(* PLC project primary, CODESYS STW CODESYS V3.5 SP11 - ESX-3CS, author Isoloader *)
(* stored: creationDateTime 2026-05-19T11:23:56.1136893, version 0.101, modificationDateTime 2026-05-14T13:26:08.1458645, organization Isoloader *)

(* {attribute 'strict'} *)
{attribute 'qualified_only'}
TYPE t_bms_fault_id : (cBMSFaultCellOverVoltageAlarmWarning := 1, cBMSFaultCellOverVoltageAlarmCritical := 2, cBMSFaultCellOverVoltageAlarmSevere := 3, cBMSFaultCellUnderVoltageAlarmWarning := 4, cBMSFaultCellUnderVoltageAlarmCritical := 5, cBMSFaultCellUnderVoltageAlarmSevere := 6, cBMSFaultCellOverDischargeAlarm := 7, cBMSFaultSystemOverVoltageAlarmWarning := 8, cBMSFaultSystemOverVoltageAlarmCritical := 9, cBMSFaultSystemOvervoltageAlarmSevere := 10, cBMSFaultSystemUnderVoltageAlarmWarning := 11, cBMSFaultSystemUnderVoltageAlarmCritical := 12, cBMSFaultSystemUnderVoltageAlarmSevere := 13, cBMSFaultCellHighTemperatureAlarmWarning := 14, cBMSFaultCellHighTemperatureAlarmCritical := 15, cBMSFaultCellHighTemperatureAlarmSevere := 16, cBMSFaultCellLowTemperatureAlarm := 17, cBMSFaultTemperatureDifferenceisTooLargeAlarmWarning := 18, cBMSFaultTemperatureDifferenceisTooLargeAlarmCritical := 19, cBMSFaultTemperatureDifferenceisTooLargeAlarmSevere := 20, cBMSFaultFireAlarm := 21, cBMSFaultPulseDischargeOverCurrentAlarmWarning := 22, cBMSFaultPulseDischargeOverCurrentAlarmCritical := 23, cBMSFaultPulseDischargeOverCurrentAlarmSevere := 24, cBMSFaultPulseRechargeOverCurrentAlarmWarning := 25, cBMSFaultPulseRechargeOverCurrentAlarmCritical := 26, cBMSFaultPulseRechargeOverCurrentAlarmSevere := 27, cBMSFaultCurrentSensorFaultAlarm := 28, cBMSFaultBMSLowVoltagePowerSupplyisAbnormalAlarm := 29, cBMSFaultSOCDifferenceisTooLargeAlarm := 30, cBMSFaultSOCJumpFaultAlarm := 31, cBMSFaultLowSOCAlarmWarning := 32, cBMSFaultLowSOCAlarmCritical := 33, cBMSFaultLowSOCAlarmSevere := 34, cBMSFaultThermalManagementSystemFaultAlarm := 35, cBMSFaultPackSelfProtectionAlarm := 37, cBMSFaultMainCircuitPrechargePrecheckFaultAlarm := 38, cBMSFaultLowInsulationInDrivingAlarmWarning := 40, cBMSFaultLowInsulationInDrivingAlarmCritical := 41, cBMSFaultLowInsulationInDrivingAlarmSevere := 42, cBMSFaultLowInsulationInChargingAlarm := 43, cBMSFaultACANCommunicationFaultAlarm := 44, cBMSFaultBMSInternalCommunicationFaultAlarm := 45, cBMSFaultBranchDisconnectedFaultAlarm := 47, cBMSFaultHVILFaultAlarm := 48, cBMSFaultMainPositiveRelayCannotbeClosedAlarm := 51, cBMSFaultMainPositiveRelayWeldedAlarm := 52, cBMSFaultMainNegativeRelayCannotbeClosedAlarm := 53, cBMSFaultMainNegativeRelayWeldedAlarm := 54, cBMSFaultChargeableEnergyStorageSystemMismatchAlarm := 72, cBMSFaultDischargingCurrentIsTooLargeInChargingAlarm := 73, cBMSFaultChargingCurrentIsTooLargeAlarm := 74, cBMSFaultFireAlarmDetectorFault := 79, cBMSFaultCellPoorConsistencyAlarm := 100, cBMSFaultSOCAlarmTooHigh := 101, cBMSFaultContinuousDischargeOvercurrentAlarmWarning := 105, cBMSFaultContinuousDischargeOvercurrentAlarmCritical := 106, cBMSFaultContinuousDischargeOvercurrentAlarmSevere := 107);
END_TYPE

(* values of t_motor_emcy_id: cEMCY_PEV_NOT_OK: change from 65499, duplicate error; cEMCY_SP_MISMATCH_XX: cEMCY_SP_MISMATCH_PUMP := 65521,//change from 65521, duplicate; cEMCY_THROTTLE_PROG: cEMCY_OPEN_COIL_EV := 65522, //duplicate id *)

(* {attribute 'strict'} *)
{attribute 'qualified_only'}
TYPE t_motor_emcy_id : (cEMCY_none := 0, cEMCY_MC_EB_COIL_SHORT := 8784, cEMCY_STBY_HIGH := 8977, cEMCY_PUMP_ZERO_EVER := 8978, cEMCY_WRONG_SET_BAT := 12544, cEMCY_WRONG_KEY_VOLT := 12545, cEMCY_VMN_HIGH := 12560, cEMCY_INIT_VMN_HIGH := 12561, cEMCY_VMN_LOW := 12576, cEMCY_INIT_VMN_LOW := 12577, cEMCY_CAPACITOR_CHARGE := 12592, cEMCY_DRIVER_SHORTED := 12817, cEMCY_CONTACTOR_DRIVER := 12833, cEMCY_EB_DRIVSHRT := 12834, cEMCY_POS_EB_SHORTED := 12835, cEMCY_EB_DRIVOPEN := 12836, cEMCY_SMARTDRIVER_KO := 13058, cEMCY_EEPROM_KO := 13840, cEMCY_THERMIC_SENS_KO := 16913, cEMCY_SENS_MOT_TEMP_KO := 17169, cEMCY_AUX_BATT_SHORT := 20481, cEMCY_EVP_COIL_OPEN := 20482, cEMCY_EVP_DRIV_SHORT := 20483, cEMCY_EVP_COIL_SHORT := 20484, cEMCY_EVP2_COIL_OPEN := 20722, cEMCY_EVP2_DRIV_SHORT := 20723, cEMCY_EVP2_COIL_SHORT := 20724, cEMCY_VKEY_OFF_SHORTED := 20737, cEMCY_LOGIC_FAILURE_1 := 20756, cEMCY_CONTACTOR_OPEN := 21569, cEMCY_CONTACTOR_CLOSED := 21570, cEMCY_WATCHDOG := 24592, cEMCY_CURRENT_GAIN := 25346, cEMCY_NO_CAN_MSG := 33072, cEMCY_NO_CAN_WR_MSGXX := 33073, cEMCY_LOGIC_FAILURE_3 := 65297, cEMCY_LOGIC_FAILURE_2 := 65298, cEMCY_PUMP_VMN_LOW := 65308, cEMCY_PUMP_VMN_HIGH := 65309, cEMCY_BATTERY_LOW := 65346, cEMCY_VACC_NOT_OK := 65358, cEMCY_INCORRECT_START := 65359, cEMCY_FORW_BACK := 65360, cEMCY_WRONG_FBSENSSET := 65361, cEMCY_PEDAL_WIRE_KO := 65366, cEMCY_BACK_EMF_HIGH := 65418, cEMCY_THERMPUSENSKO := 65419, cEMCY_1175_NOT_ACTIVE := 65420, cEMCY_STO_SS1_ACTIVEXX := 65421, cEMCY_STO_SS1_ALARM_XX := 65422, cEMCY_SAFETY_INIT_XX := 65423, cEMCY_SAFETY_WARN_XX := 65424, cEMCY_SAFETY_SW_XX := 65425, cEMCY_SAFETY_DIAG_XX := 65426, cEMCY_BMS_FAULT := 65427, cEMCY_BMS_NOT_READY := 65428, cEMCY_WRONG_PERFORM := 65429, cEMCY_NO_CAN_MSG_DISP := 65430, cEMCY_POT_MISMATCH := 65431, cEMCY_SENSOR_SUPPLY_XX := 65432, cEMCY_OFFSET_SPDSENS := 65433, cEMCY_AGV := 65434, cEMCY_REMA_T_ALARM := 65436, cEMCY_FAULT_DRVPOWER := 65437, cEMCY_NOT_RDY_DRVPOW := 65438, cEMCY_HVIL_FAIL := 65439, cEMCY_SENS_BAT_TEMP_KO := 65440, cEMCY_RPM_HIGH := 65441, cEMCY_POSEBSHORT_PIN := 65442, cEMCY_ED_SLIP_MISMATCH := 65443, cEMCY_POSEBSHORT_GND := 65444, cEMCY_SHORT_CIRCUIT_KO := 65445, cEMCY_SHORT_CIRCUIT := 65446, cEMCY_IMS_ERROR := 65447, cEMCY_SPEED_FBERR_XX := 65448, cEMCY_EMERGENCY := 65449, cEMCY_SPEED_OVERHEAD := 65455, cEMCY_COIL_SHOR_EB := 65457, cEMCY_MOTOR_TEMP_STOP := 65458, cEMCY_STEER_SENSOR_KO := 65459, cEMCY_OVERLOAD := 65460, cEMCY_EVP2_DRIVER_OPEN := 65464, cEMCY_TILLER_ERROR := 65465, cEMCY_LIFT_LOWER := 65467, cEMCY_PUMP_VACC_NOT_OK := 65468, cEMCY_PUMP_INC_START := 65469, cEMCY_PUMP_VMN_NOT_OK := 65470, cEMCY_PUMP_I_NO_ZERO := 65471, cEMCY_PUMP_VACC_RANGE := 65472, cEMCY_MOTPHASE_SH := 65476, cEMCY_WRONG_SLAVE_VER := 65477, cEMCY_MS_PAR_CHK_MISM := 65478, cEMCY_PARAM_TRANSFER := 65479, cEMCY_VDC_OFF_SHORTED := 65480, cEMCY_CURRENT_PROFILE := 65481, cEMCY_VDC_LINK_OVERV := 65482, cEMCY_HW_FAULT_MC := 65483, cEMCY_BRAKE_RUN_OUT := 65484, cEMCY_EPS_RELAY_OPEN := 65485, cEMCY_WRONG_RAM_MEM := 65490, cEMCY_STALL_ROTOR := 65491, cEMCY_POWER_MISMATCH := 65492, cEMCY_WSET_TG_EB_XX := 65492, cEMCY_INPUT_MISMATCH := 65493, cEMCY_POSITIVE_LC_OPEN := 65493, cEMCY_EB_COIL_OPEN := 65496, cEMCY_PEB_PEVP_NOT_OK := 65499, cEMCY_PEV_NOT_OK := 65500, cEMCY_HANDBRAKE := 65501, cEMCY_SEAT_MISMATCH := 65502, cEMCY_VACC_OUT_RANGE := 65506, cEMCY_HW_FAULT := 65507, cEMCY_OUT_MISMATCH_XX := 65507, cEMCY_HW_FAULT_EB := 65509, cEMCY_LC_COIL_OPEN := 65510, cEMCY_CONT_DRV_EV := 65512, cEMCY_POWERMOS_SHORTED := 65513, cEMCY_CTRAP_THRESHOLD := 65515, cEMCY_HW_FAULT_EV := 65518, cEMCY_CONTROLLER_MISM := 65519, cEMCY_OUT_MISMATCH_PU := 65520, cEMCY_COIL_SHOR_EVAUX := 65521, cEMCY_SP_MISMATCH_XX := 65522, cEMCY_THROTTLE_PROG := 65523, cEMCY_IQ_MISMATCHED := 65525, cEMCY_EVP_DRIVER_OPEN := 65528, cEMCY_DRV_SHOR_EV := 65529, cEMCY_ANALOG_INPUT := 65530, cEMCY_FIELD_ORIENT_KO := 65533);
END_TYPE

TYPE t_radio_emcy_id : (cEMCY_none := 0, cEMCY_CAN_OVERRUN := 33040, cEMCY_CAN_IN_ERROR_PASSIVE_MODE := 33056, cEMCY_LIFE_GUARD_ERROR_OR_HEARTBEAT_ERROR := 33072, cEMCY_RECOVERED_FROM_BUS_OFF := 33088, cEMCY_TRANSMIT_COB_ID_COLLISION := 33104, cEMCY_PDO_NOT_PROCESSED_DUE_TO_LENGTH_ERROR := 33296, cEMCY_PDO_LENGTH_EXCEEDED := 33312, cEMCY_GENERIC_ERROR := 4096, cEMCY_CURRENT := 8192, cEMCY_CURRENT_DEVICE_INPUT_SIDE := 8448, cEMCY_CURRENT_INSIDE_THE_DEVICE := 8704, cEMCY_CURRENT_DEVICE_OUTPUT_SIDE := 8960, cEMCY_CURRENT_AT_OUTPUTS_TOO_HIGH := 8976, cEMCY_SHORT_CIRCUIT_AT_OUTPUTS := 8992, cEMCY_LOAD_DUMP_AT_OUTPUTS := 9008, cEMCY_VOLTAGE := 12288, cEMCY_MAINS_VOLTAGE := 12544, cEMCY_INPUT_VOLTAGE_TOO_HIGH := 12560, cEMCY_INPUT_VOLTAGE_TOO_LOW := 12576, cEMCY_VOLTAGE_INSIDE_THE_DEVICE := 12800, cEMCY_INTERNAL_VOLTAGE_TOO_HIGH := 12816, cEMCY_INTERNAL_VOLTAGE_TOO_LOW := 12832, cEMCY_OUTPUT_VOLTAGE := 13056, cEMCY_OUTPUT_VOLTAGE_TOO_HIGH := 13072, cEMCY_OUTPUT_VOLTAGE_TOO_LOW := 13088, cEMCY_TEMPERATURE := 16384, cEMCY_AMBIENT_TEMPERATURE := 16640, cEMCY_DEVICE_TEMPERATURE := 16896, cEMCY_DEVICE_HARDWARE := 20480, cEMCY_DEVICE_SOFTWARE := 24576, cEMCY_INTERNAL_SOFTWARE := 24832, cEMCY_USER_SOFTWARE := 25088, cEMCY_DATA_SET := 25344, cEMCY_ADDITIONAL_MODULES := 28672, cEMCY_MONITORING := 32768, cEMCY_COMMUNICATION := 33024, cEMCY_PROTOCOL_ERROR := 33280, cEMCY_EXTERNAL_ERROR := 36864, cEMCY_ADDITIONAL_FUNCTIONS := 61440, cEMCY_DEVICE_SPECIFIC := 65280);
END_TYPE

TYPE t_functional_diagnostic : (cFunctionalDiagnosticOK := 0, cFunctionalDiagnosticNotYetActive := 1, cFunctionalDiagnosticNotEnabled := 2, cFunctionalDiagnosticNotStationary := 3, cFunctionalDiagnosticWaitingOnPreviousToExit := 4, cFunctionalDiagnosticWaitingToExit := 5, cFunctionalDiagnosticRace := 6);
END_TYPE

(* {attribute 'qualified_only'} *)
TYPE t_mode_state : (cModeStateInactive := 0, cModeStateEntering := 1, cModeStateExiting := 2, cModeStateActive := 3);
END_TYPE

TYPE t_pmc_set : ARRAY[1..32] OF t_prog_mov_code;
END_TYPE

TYPE t_prog_mov_diagnostic : (cProgMovDiagnosticDisabled := 0, cProgMovDiagnosticEnabling := 1, cProgMovDiagnosticPrepared := 2, cProgMovDiagnosticActivating := 3, cProgMovDiagnosticWaiting := 4, cProgMovDiagnosticStarting := 5, cProgMovDiagnosticRunning := 6, cProgMovDiagnosticFinishing := 7, cProgMovDiagnosticInterrupted := 8, cProgMovDiagnosticLeaving := 9, cProgMovDiagnosticDeactivatingFromWaiting := 10, cProgMovDiagnosticDeactivatingFromRunning := 11, cProgMovDiagnosticDeactivatingFromFinished := 12, cProgMovDiagnosticDeactivatingFromLeaving := 13, cProgMovDiagnosticInactiveTimeout := 14);
END_TYPE

TYPE t_slew_state : STRUCT
  targetAngle : REAL;
  wheelVelocityFactor : REAL;
  steerInput : REAL;
END_STRUCT;
END_TYPE

TYPE t_steer_mode_diagnostic : (cSteerModeDiagnosticOK := 0, cSteerModeDiagnosticNotEnabled := 1, cSteerModeDiagnosticUnableToLockDrive := 2, cSteerModeDiagnosticChanging := 3);
END_TYPE

TYPE t_direction : (cDirectionStationary := 0, cDirectionForward := 1, cDirectionReverse := 2);
END_TYPE

(* values of t_motor_diagnostic: cMotorDiagnosticHoldStationary: cMotorDiagnosticControllerTemperature := 9, cMotorDiagnosticMotorTemperature := 10, *)

TYPE t_motor_diagnostic : (cMotorDiagnosticOK := 0, cMotorDiagnosticDisabled := 2, cMotorDiagnosticActiveDisallow := 3, cMotorDiagnosticNotOperational := 4, cMotorDiagnosticOperatingMode := 6, cMotorDiagnosticStalled := 7, cMotorDiagnosticHunting := 8, cMotorDiagnosticHoldStationary := 11, cMotorDiagnosticInitializeHold := 12);
END_TYPE

TYPE t_movement_diagnostic : (cMovementDiagnosticOK := 0, cMovementDiagnosticInterlock := 1, cMovementDiagnosticDisabled := 2, cMovementDiagnosticActiveDisallow := 3, cMovementDiagnosticNotOperational := 4, cMovementDiagnosticUMFS := 5, cMovementDiagnosticOperatingMode := 6, cMovementDiagnosticFunctionalMode := 7, cMovementDiagnosticStalled := 8, cMovementDiagnosticHunting := 9, cMovementDiagnosticDerived := 10, cMovementDiagnosticBrakeEngaged := 11, cMovementDiagnosticBrakeDisengaged := 12, cMovementDiagnosticSteeringModeChange := 13, cMovementDiagnosticSteeringState := 14, cMovementDiagnosticDeadband := 15, cMovementDiagnosticThreshold := 16);
END_TYPE

TYPE t_stall_recovery : (cStallRecoveryNone := 0, cStallRecoveryDone := 1, cStallRecoveryWait := 2, cStallRecoveryReverse := 3);
END_TYPE

TYPE t_stall_state : (cStallStateNone := 0, cStallStateDetected := 1, cStallStateCurrent := 2, cStallStateClearing := 3);
END_TYPE

VAR_GLOBAL CONSTANT  (* GlobalVariablesPeripheralPLC *)
  cRCSoftware : USINT := 0;
  cRCConfiguration : USINT := 1;
  cRCVBBS : USINT := 2;
  cRCVBB1 : USINT := 3;
  cRCVBB2 : USINT := 4;
  cRCPLCTemp : USINT := 5;
END_VAR

VAR_GLOBAL CONSTANT  (* GlobalVariablesPrimary *)
  cSteerMotorMaximumVelocityAsHz : REAL := 50.0;
  cTransMotorMaximumVelocityAsHz : REAL := 55.0;
  gSystemPrimary : REFERENCE TO SystemPrimary;
  gBMSASupplementaryCommand : USINT := 0;  (* foobar *)
  gBMSASupplementaryState : USINT := 0;
  gBMSBSupplementaryCommand : USINT := 0;
  gBMSBSupplementaryState : USINT := 0;
  sCommandZero : t_command_definition := (command := cTokenZero);
  sCommandUpper : t_command_definition := (command := sTokenUpper);
END_VAR

FUNCTION_BLOCK PLCPrimary EXTENDS PLC
  VAR CONSTANT
    cBackupBatteryVoltageMin : REAL := 22.0;
    cMBTemperatureMax : REAL := 75.0;
    cCPUTemperatureMax : REAL := 80.0;
    cWatchdogMaxNormal : UINT := 500;  (* units of 0.5ms *)
    cWatchdogMaxDebug : UINT := 8000;  (* units of 0.5ms *)
  END_VAR
  VAR
    lVRTriggerRestartPLC : ValueReferenceBool;
    lTriggerRestartPLC : BOOL;
    lVRTriggerRestartSupervisor : ValueReferenceBool;
    lTriggerRestartSupervisor : BOOL;
    lVREnableMaintenanceSwitch : ValueReferenceBool;
    lEnableMaintenanceSwitch : BOOL := FALSE;
    lOutputStayAlive : ValueObjectBoolOutputReferenceUSINTAsBool;
    lOutputMainRelay : ValueObjectBoolOutputReferenceUSINTAsBool;
    lInputIgnition : ValueObjectBoolInputReferenceUSINTAsBool;
    lInputMaintenance : ValueObjectBoolInputReferenceDINTAsBool;
    lAlarmBackupBatteryVoltageLow : ReportableAlarmAllowableUp;
    lAlarmDeviceTemperature : ReportableAlarm;
    lVoltage : FB_x_sys_get_adc_value_scaled;
    lMBTemperature : FB_x_sys_get_temperature;
    lCPUTemperature : FB_x_sys_get_temperature;
    lSysClose : FB_x_sys_close;
    lSystemInfo : FB_x_sys_get_system_information;
    lSupervisor : FB_x_ssv_init;
    lSupervisorStatus : FB_x_ssv_get_status;
    lWatchdogTrigger : FB_x_ssv_trigger;
    lWatchdogTriggerState : FB_x_ssv_set_trigger;
    lPreviousShutdownBySupervisor : BOOL;
  END_VAR

            ;
          

METHOD setWatchdogDisabled
                  lSupervisor.ot_SupervisorConfig.u16_WDmax := 0;
lSupervisor();
                
END_METHOD

METHOD initialize
  VAR
    i : USINT;
  END_VAR
                  Name := 'PLC';

lVRTriggerRestartPLC.initializeValueReference(lTriggerRestartPLC,NopSelf,'RestartPLC','Trigger a restart of the PLC','',cValueStyleTrigger);
lVRTriggerRestartSupervisor.initializeValueReference(lTriggerRestartSupervisor,NopSelf,'RestartSuperv','Trigger a restart of the supervisor','',cValueStyleTrigger);
lVREnableMaintenanceSwitch.initializeValueReference(lEnableMaintenanceSwitch,NopSelf,'EnblMaintSwitch','Maintenance switch is enabled','',cValueStyleParameter);

lOutputStayAlive.initializeValueObjectOp(OpSelf,'oStayAlive','The stay-alive output','',cValueStyleConfigurable);
lOutputMainRelay.initializeValueObjectOp(OpSelf,'oMainRelay','The main relay output','',cValueStyleConfigurable);

lInputIgnition.initializeValueObjectOp(OpSelf,'iIgnition','The ignition input','',cValueStyleConfigurable);
lInputMaintenance.initializeValueObjectOp(OpSelf,'iMaintenance','The maintenance switch input','',cValueStyleConfigurable);

lAlarmBackupBatteryVoltageLow.initializeState(NopSelf,'',cACBackupBatteryVoltageLow);
lAlarmBackupBatteryVoltageLow.AllowableSystemState := cSystemStateStandby;
lAlarmBackupBatteryVoltageLow.UpperSystemStateScope := cSystemStateStandby;
lAlarmBackupBatteryVoltageLow.LowerSystemStateScope := cSystemStateStandby;
lAlarmBackupBatteryVoltageLow.Life := 10;
lAlarmBackupBatteryVoltageLow.InitialSeverity := cSeverityNone;
lAlarmBackupBatteryVoltageLow.SeverityWarningTimeout := T#250MS;
lAlarmBackupBatteryVoltageLow.SeverityErrorTimeout := T#30S;
lAlarmBackupBatteryVoltageLow.SeverityCriticalTimeout := T#300S;
lAlarmBackupBatteryVoltageLow.ForceTrigger := true;

lAlarmDeviceTemperature.initializeState(NopSelf,'',cACDeviceTemperature);

SUPER^.initialize();
SubSystem := cSubsystemPowerpack;

lSupervisor.ot_SupervisorConfig.u16_WDmin := 0;
lSupervisor.ot_SupervisorConfig.u8_UEmin := 32;
lSupervisor.ot_SupervisorConfig.u8_UEmax := 140;
lSupervisor.ot_SupervisorConfig.u8_Reset := X_SSV_ERR_WD_USER;
setWatchdog();

lSupervisorStatus();
lPreviousShutdownBySupervisor := (UDINT_TO_BOOL(lSupervisorStatus.ot_SupervisorStatus.u32_LastReset AND X_SSV_CPURST_WD_USER));
IF (lPreviousShutdownBySupervisor) THEN
	lPreviousShutdownCode := MAX(lPreviousShutdownCode,t_shutdown_code.cShutdownCodeSupervisor);
END_IF

lWatchdogTrigger.ou16_TriggerType := X_SSV_TRIGGER;
lWatchdogTrigger();

lSystemInfo();
IF (lSystemInfo.ot_SysInfo.t_LastTrap.u32_Address<>0) THEN
	lPreviousShutdownCode := MAX(lPreviousShutdownCode,t_shutdown_code.cShutdownCodeTrapDetected);
	lTrapDetected := FALSE;
END_IF

// generally the case for systems where power and ignition are tied foobar
IF (lPreviousShutdownCode=t_shutdown_code.cShutdownCodeUnknown) THEN
	lPreviousShutdownCode := t_shutdown_code.cShutdownCodeIgnition;
END_IF

lVoltage.ou16_Channel := X_SYS_ADC_U_UB1;
lMBTemperature.ou16_Channel := X_SYS_TEMP_BOARD;
lCPUTemperature.ou16_Channel := X_SYS_TEMP_CPU;

lOutputStayAlive.Value := TRUE;
lOutputMainRelay.Value := TRUE;

                
END_METHOD

METHOD operator
                  SUPER^.operator();

lWatchdogTriggerState.ou16_TriggerState := BOOL_TO_UINT(NOT(UINT_TO_BOOL(lWatchdogTriggerState.ou16_TriggerState)));
lWatchdogTriggerState();
lWatchdogTrigger();

IF (NOT(lInputIgnition.Value)) THEN
	lShutdownCode.Value := t_shutdown_code.cShutdownCodeIgnition;
	lSysClose();	
END_IF

IF (lTriggerRestartPLC) THEN
	lTriggerRestartPLC := FALSE;

	lShutdownCode.Value := t_shutdown_code.cShutdownCodeSoftware;
  	lSysClose();
END_IF

IF (lTriggerRestartSupervisor) THEN
	lTriggerRestartSupervisor := FALSE;
	lSupervisor();
END_IF

lVoltage();
IF (Voltage<cBackupBatteryVoltageMin) THEN
	lAlarmBackupBatteryVoltageLow.test(FALSE);
END_IF

IF ((MBTemperature>cMBTemperatureMax) OR
	(CPUTemperature>cCPUTemperatureMax)) THEN
	lAlarmDeviceTemperature.trigger(FALSE);
END_IF



                
END_METHOD

METHOD initializePLC
  VAR_INPUT
    outputStayAlive : REFERENCE TO USINT;
    outputMainRelay : REFERENCE TO USINT;
    inputIgnition : REFERENCE TO USINT;
    inputMaintenance : REFERENCE TO DINT;
  END_VAR
                  lOutputStayAlive.OutputReference REF= outputStayAlive;
lOutputMainRelay.OutputReference REF= outputMainRelay;

lInputIgnition.InputReference REF= inputIgnition;
lInputMaintenance.InputReference REF= inputMaintenance;

                
END_METHOD

METHOD setWatchdogDebug
                  lSupervisor.ot_SupervisorConfig.u16_WDmax := cWatchdogMaxDebug;
lSupervisor();

                
END_METHOD

METHOD setWatchdogNormal
                  lSupervisor.ot_SupervisorConfig.u16_WDmax := cWatchdogMaxNormal;
lSupervisor();

                
END_METHOD

PROPERTY MBTemperature : REAL
GET
                    MBTemperature := INT_TO_REAL(lMBTemperature.os16_Value)/10.0;

                  
END_GET
END_PROPERTY

PROPERTY Voltage : REAL
GET
                    Voltage := DINT_TO_REAL(lVoltage.os32_Value)/1000.0;

                  
END_GET
END_PROPERTY

PROPERTY CPUTemperature : REAL
GET
                    CPUTemperature := INT_TO_REAL(lCPUTemperature.os16_Value)/10.0;

                  
END_GET
END_PROPERTY

PROPERTY MaintenanceMode : BOOL
GET
                    MaintenanceMode := (((lEnableMaintenanceSwitch) AND (lInputMaintenance.Value))
	OR (lMaintenanceMode));
                  
END_GET
END_PROPERTY
END_FUNCTION_BLOCK

FUNCTION_BLOCK BMS EXTENDS OutputSystemStateAuto
  VAR CONSTANT
    cBMSCurrentMax : REAL := 900;
    cBMSChargeSafetyMargin : REAL := 0.0;
    cBMSChargeDerateFactor : REAL := 1.0;
    cBMSDishargeSafetyMargin : REAL := 0.0;
    cBMSDishargeDerateFactor : REAL := 1.0;
    cRetryPeriod : t_time := TIME#1m0s0ms;
    cBMSSOCWarningLow : t_percentage := 0.15;
    cBMSSOCOperatingMinimum : t_percentage := 0.05;
    cBMSSOCStandbyMinimum : t_percentage := 0.02;
    cSOCRecoveryPeriod : t_time := TIME#1m0s0ms;
    cSOCRecoveryChargingCurrentMinimum : REAL := -1.0;
  END_VAR
  VAR
    lVREnableSOCRecoveryMode : ValueReferenceBool;
    lEnableSOCRecoveryMode : BOOL := FALSE;
    lVRTriggerSOCRecoveryTimer : ValueReferenceBool;
    lTriggerSOCRecoveryTimer : BOOL := FALSE;
    lVREnableRestart : ValueReferenceBool;
    lEnableRestart : BOOL := TRUE;
    lVRRestartCount : ValueReferenceUSINT;
    lRestartCount : USINT := 0;
    lVRDisableConnect : ValueReferenceBool;
    lDisableConnect : BOOL := FALSE;
    lVRSOCRecoveryChargingCurrentMinimum : ValueReferenceReal;
    lSOCRecoveryChargingCurrentMinimum : REAL := cSOCRecoveryChargingCurrentMinimum;
    lVREnableBMS : ValueReferencePersistentUINT;
    lEnableBMS : PersistentUINT;
    lAlarmBMSNotConnected : ReportableAlarmAllowableUp;
    lAlarmSOCBelowOperatingMinimum : ReportableSystemControl;
    lAlarmSOCBelowStandbyMinimum : ReportableAlarm;
    lAlarmBMSAvailabilityInsufficient : ReportableSystemControl;
    lAlarmSOCWarningLow : ReportableAlarm;
    lAlarmBMSAvailabilityLimited : ReportableAlarmEscalating;
    lAlarmBMSFailToConnect : ReportableAlarm;
    lAlarmChargeCutback : ReportableChargeModulation;
    lAlarmDischargeCutback : ReportableChargeModulation;
    lTimer : t_timer;
    lBMSStandbyState : t_bms_state := cBMSStateStandby;
    lRequestedState : t_bms_state;
    lCurrentState : t_bms_state;
    lAvailability : t_percentage;
    lVRAvailability : ValueReferencePercentage;
    lAvailabilityMinimum : t_percentage := 1.0;
    lRequestedBMSChargeState : t_bms_charge_state;
    lCurrentBMSChargeState : t_bms_charge_state;
    lRequestedTMSState : t_tms_state;
    lCurrentTMSState : t_tms_state;
    lBalancing : BOOL;
    lSOC : t_percentage;
    lVRSOC : ValueReferencePercentage;
    lSOCMin : t_percentage;
    lSOCMax : t_percentage;
    lVoltage : REAL;
    lVRVoltage : ValueReferenceReal;
    lVoltageMin : REAL;
    lVoltageMax : REAL;
    lCurrent : REAL;
    lVRCurrent : ValueReferenceReal;
    lCurrentMin : REAL;
    lCurrentMax : REAL;
    lChargeCurrentLimit : REAL;
    lDischargeCurrentLimit : REAL;
    lChargingCurrentTarget : REAL;
    lChargingVoltageTarget : REAL;
    lRequestedCoolantTemperature : REAL;
    lCurrentCoolantTemperature : REAL;
    lCurrentLevel : t_percentage;  (* foostrip lDischargePower: REAL; lDischargeCumulativeEnergy: REAL; lChargePower: REAL; lChargeCumulativeEnergy: REAL; *)
    lCurrentExceeding : REAL;
    lCurrentDerateScaling : REAL;
    lChargeCurrent : REAL;
    lChargeSafetyMargin : REAL := cBMSChargeSafetyMargin;
    lChargeDerateFactor : REAL := cBMSChargeDerateFactor;
    lChargeDerate : t_percentage;
    lDischargeCurrent : REAL;
    lDischargeSafetyMargin : REAL := cBMSDishargeSafetyMargin;
    lDischargeDerateFactor : REAL := cBMSDishargeDerateFactor;
    lDischargeDerate : t_percentage;
    lRetryTimer : t_timer;
    lRestartCountMax : USINT := 2;
    lSOCRecoveryTimer : t_timer;
  END_VAR

            ;
          

METHOD currentDerating
                  lCurrentLevel := lCurrent/cBMSCurrentMax;

lChargeCurrentLimit := ABS(lChargeCurrentLimit);
IF (lChargeCurrent>0.0) THEN
	lCurrentExceeding := MAX(lChargeCurrent-lChargeCurrentLimit+lChargeSafetyMargin,0.0);
	lCurrentDerateScaling := lCurrentExceeding/lChargeCurrent*lChargeDerateFactor;
	lChargeDerate := MIN(MAX((1.0 - lCurrentDerateScaling),0.0),1.0);
ELSE
	lChargeDerate := 1.0;
END_IF

IF (ABS(lChargeDerate)<1.0) THEN
	lAlarmChargeCutback.ScalingCharge := lChargeDerate;
	lAlarmChargeCutback.trigger(FALSE);
END_IF

lDischargeCurrentLimit := ABS(lDischargeCurrentLimit);
IF (lDischargeCurrent>0.0) THEN
	lCurrentExceeding := MAX(lDischargeCurrent-lDischargeCurrentLimit+lDischargeSafetyMargin,0.0);
	lCurrentDerateScaling := lCurrentExceeding/lDischargeCurrent*lDischargeDerateFactor;
	lDischargeDerate := MIN(MAX((1.0 - lCurrentDerateScaling),0.0),1.0);
ELSE
	lDischargeDerate := 1.0;
END_IF

IF (ABS(lDischargeDerate)<1.0) THEN
	lAlarmDischargeCutback.ScalingDischarge := lDischargeDerate;
	lAlarmDischargeCutback.trigger(FALSE);
END_IF
                
END_METHOD

METHOD _operatorNull
                  lCurrentBMSChargeState := cBMSChargeStateShutdown;
lRequestedTMSState := cTMSStateShutdown;
lRequestedCoolantTemperature := 30.0;

lBalancing := FALSE;

lChargeCurrent := 0.0;
lDischargeCurrent := 0.0;

lChargeCurrentLimit := 0.0;
lDischargeCurrentLimit := 0.0;
	
lChargingCurrentTarget := 0.0;
lChargingVoltageTarget := 0.0;

//lDischargePower := lControllerBMSA.DischargePower;
//lDischargeCumulativeEnergy := lControllerBMSA.DischargeCumulativeEnergy;
//lChargePower := lControllerBMSA.ChargePower;
//lChargeCumulativeEnergy := lControllerBMSA.ChargeCumulativeEnergy;

                
END_METHOD

METHOD initialize
                  lVRCurrent.initializeValueReference(lAvailability,NopSelf,'Current','Battery system current','amps',cValueStyleConfigurable);
lVRSOC.initializeValueReference(lAvailability,NopSelf,'SOC','Battery system SOC','',cValueStyleConfigurable);
lVRVoltage.initializeValueReference(lAvailability,NopSelf,'Voltage','Battery system voltage','volts',cValueStyleConfigurable);
lVRAvailability.initializeValueReference(lAvailability,NopSelf,'Availability','Battery system availability','',cValueStyleConfigurable);
	
lVREnableSOCRecoveryMode.initializeValueReference(lEnableSOCRecoveryMode,NopSelf,'EnblSOCRecovery','Enable recovery from low SOC','',cValueStyleParameter);
lVRTriggerSOCRecoveryTimer.initializeValueReference(lTriggerSOCRecoveryTimer,NopSelf,'SOCRecTimRst','Trigger low SOC recovery timer','',cValueStyleTrigger);
lVREnableRestart.initializeValueReference(lEnableRestart,NopSelf,'EnblRestart','Enable restart of battery system','',cValueStyleParameter);
lVRRestartCount.initializeValueReference(lRestartCount,NopSelf,'RestartCount','Battery system restart attempt count','',cValueStyleConfigurable);
lVRDisableConnect.initializeValueReference(lDisableConnect,NopSelf,'DsblConnect','Disable battery system contactors','',cValueStyleParameter);
lVRSOCRecoveryChargingCurrentMinimum.initializeValueReference(lSOCRecoveryChargingCurrentMinimum,NopSelf,'SOCRecCurrMin','Low SOC recovery charging current','',cValueStyleParameter);

lVREnableBMS.initializeValueReference(lEnableBMS,NopSelf,'EnblBMS','Enable battery system','',cValueStyleParameter);
lEnableBMS.Identifier := t_persistent_id.cPersistentID_EnableBMS;
lEnableBMS.initialize();

lAlarmBMSAvailabilityInsufficient.initializeState(NopSelf,'',cACBMSAvailabilityInsufficient);
lAlarmBMSAvailabilityInsufficient.Control := cSystemControlStop;
lAlarmBMSAvailabilityInsufficient.AllowableSystemState := cSystemStateCharging;

lAlarmSOCBelowOperatingMinimum.initializeState(NopSelf,'',cACSOCBelowOperatingMinimum);
lAlarmSOCBelowOperatingMinimum.Control := cSystemControlStop;
lAlarmSOCBelowOperatingMinimum.AllowableSystemState := cSystemStateCharging;

lAlarmSOCBelowStandbyMinimum.initializeState(NopSelf,'',cACSOCBelowStandbyMinimum);

lAlarmBMSNotConnected.initializeState(NopSelf,'',cACBMSNotConnected);
lAlarmBMSNotConnected.AllowableSystemState := cSystemStatePreparing;
lAlarmBMSNotConnected.UpperSystemStateScope := cSystemStatePreparing;
lAlarmBMSNotConnected.LowerSystemStateScope := cSystemStatePreparing;
lAlarmBMSNotConnected.Life := 10;
lAlarmBMSNotConnected.InitialSeverity := cSeverityNone;
lAlarmBMSNotConnected.SeverityWarningTimeout := T#5S;
lAlarmBMSNotConnected.SeverityErrorTimeout := T#20S;
lAlarmBMSNotConnected.SeverityCriticalTimeout := T#60S;

lAlarmChargeCutback.initializeState(NopSelf,'',cACBMSChargeCutback);
lAlarmChargeCutback.Qualifier := cChargeQualifierCharge;
lAlarmChargeCutback.registerServer(gSystemPrimary.Travel.ChargeInterlock);
lAlarmChargeCutback.registerServer(gSystemPrimary.Lift.ChargeInterlock);

lAlarmDischargeCutback.initializeState(NopSelf,'',cACBMSDischargeCutback);
lAlarmDischargeCutback.Qualifier := cChargeQualifierDischarge;
lAlarmDischargeCutback.registerServer(gSystemPrimary.Travel.ChargeInterlock);
lAlarmDischargeCutback.registerServer(gSystemPrimary.Lift.ChargeInterlock);

lAlarmSOCWarningLow.initializeState(NopSelf,'',cACSOCWarningLow);
lAlarmSOCWarningLow.Life := 100;

lAlarmBMSFailToConnect.initializeState(NopSelf,'',cACBMSFailToConnect);

lAlarmBMSAvailabilityLimited.initializeState(NopSelf,'',cACBMSAvailabilityLimited);
lAlarmBMSAvailabilityLimited.Life := 10;
lAlarmBMSAvailabilityLimited.InitialSeverity := cSeverityNone;
lAlarmBMSAvailabilityLimited.SeverityWarningTimeout := T#30S;
lAlarmBMSAvailabilityLimited.SeverityErrorTimeout := T#60S;
lAlarmBMSAvailabilityLimited.SeverityCriticalTimeout := T#120S;

SUPER^.initialize();
SubSystem := cSubsystemBattery;

lTimer.initialize();

lOutputSystemState := cSystemStatePreparing;

lRetryTimer.initialize();
lRetryTimer.Enable := TRUE;
lRetryTimer.Period := cRetryPeriod;

lSOC := 0.0;

lSOCRecoveryTimer.initialize();
lSOCRecoveryTimer.Enable := TRUE;
lSOCRecoveryTimer.Period := cSOCRecoveryPeriod;

// recovery software: to prevent BMS system from starting up when backup battery is failing and battery precharge is resetting plc due to low secondary voltage
// lOutput.ManualOverrideValue := TRUE;
// lOutput.OverrideValue := false;
                
END_METHOD

METHOD operator
                  lOutput.Value := ((gSystemPrimary.SystemState.State>=lOutputSystemState) AND
	(gSystemPrimary.UInterface.EnableBatteryPack));

SUPER^.operator();

IF ((gSystemPrimary.SystemState.State>cSystemStateStandby) AND (Availability<1.0)) THEN
	lAlarmBMSAvailabilityLimited.trigger(FALSE);
END_IF

IF ((gSystemPrimary.SystemState.State>cSystemStatePreparing) AND (Availability<lAvailabilityMinimum)) THEN
	lAlarmBMSAvailabilityInsufficient.trigger(FALSE);
END_IF

IF (lSOCMin<cBMSSOCWarningLow) THEN
	lAlarmSOCWarningLow.trigger(FALSE);
END_IF

IF (lSOCMin<cBMSSOCOperatingMinimum) THEN
	lAvailability := 0.0;
	lAlarmSOCBelowOperatingMinimum.trigger(FALSE);
END_IF

IF (lSOCMin<cBMSSOCStandbyMinimum) THEN		
	IF (gSystemPrimary.SystemState.State<cSystemStateStandby) THEN
		lSOCRecoveryTimer.reset();
	END_IF
	
	IF (lTriggerSOCRecoveryTimer) THEN
		lTriggerSOCRecoveryTimer := FALSE;
		lSOCRecoveryTimer.reset();
	END_IF

	IF (lCurrent<lSOCRecoveryChargingCurrentMinimum) THEN
		lSOCRecoveryTimer.reset();
	END_IF

	lSOCRecoveryTimer.operator();

	IF (lSOCRecoveryTimer.Expired) THEN
		lAlarmSOCBelowStandbyMinimum.trigger(FALSE);

		IF (NOT(lEnableSOCRecoveryMode)) THEN
			gSystemPrimary.SystemState.transitionForceMax(cSystemStateStandby,ADR(lAlarmSOCBelowStandbyMinimum),lAlarmSOCBelowStandbyMinimum.Override);
		END_IF
	END_IF
ELSE
	lSOCRecoveryTimer.reset();
END_IF

(* wait until connected *)
IF (lCurrentState<>cBMSStateConnected) THEN
	lAlarmBMSNotConnected.test(FALSE);
END_IF

currentDerating();

lRequestedState := lBMSStandbyState;

IF ((gSystemPrimary.SystemState.State>=lOutputSystemState) AND
	(gSystemPrimary.UInterface.EnableBatteryPack)) THEN
	
	IF (lDisableConnect) THEN
		lRequestedState := cBMSStateDisconnected;
	ELSE		
		lRequestedState := cBMSStateConnected;

		lRetryTimer.operator();
		IF ((lRetryTimer.Expired) AND
			(lCurrentState<>cBMSStateConnected) AND
			(lEnableRestart)) THEN

			lAlarmBMSFailToConnect.trigger(FALSE);

			IF (lRestartCount<lRestartCountMax) THEN
				(*IF (lCurrentState>cBMSStateShutdown) THEN
					cycleStandby();
				ELSE
					cycleOutputOff();
				END_IF*)
			
				cycleOutput();

				lRestartCount := lRestartCount + 1;
				lRetryTimer.reset();
			END_IF
		END_IF
	END_IF
ELSE
	lRetryTimer.reset();
	lRestartCount := 0;
	//	consider lSOCRecoveryTimer.reset(); //foobar
END_IF

                
END_METHOD

METHOD resetSOCRecovery
                  lSOCRecoveryTimer.reset();

lRestartCount := 0;
lRetryTimer.reset();
                
END_METHOD

METHOD cycleStandby
                  
                
END_METHOD

PROPERTY Availability : t_percentage
GET
                    Availability := lAvailability;
                  
END_GET
END_PROPERTY

PROPERTY AvailabilityMinimum : t_percentage
GET
                    AvailabilityMinimum := lAvailabilityMinimum;
                  
END_GET
SET
                    lAvailabilityMinimum := AvailabilityMinimum;
                  
END_SET
END_PROPERTY

PROPERTY Balancing : BOOL
GET
                    Balancing := lBalancing;

                  
END_GET
END_PROPERTY

PROPERTY ChargeCurrent : REAL
GET
                    ChargeCurrent := lChargeCurrent;

                  
END_GET
END_PROPERTY

PROPERTY ChargeCurrentLimit : REAL
GET
                    ChargeCurrentLimit := lChargeCurrentLimit;

                  
END_GET
END_PROPERTY

PROPERTY ChargeDerate : t_percentage
GET
                    ChargeDerate := lChargeDerate;
                  
END_GET
END_PROPERTY

PROPERTY ChargingCurrentTarget : REAL
GET
                    ChargingCurrentTarget := lChargingCurrentTarget;

                  
END_GET
END_PROPERTY

PROPERTY ChargingVoltageTarget : REAL
GET
                    ChargingVoltageTarget := lChargingVoltageTarget;

                  
END_GET
END_PROPERTY

(* {attribute 'monitoring' := 'call'} *)
PROPERTY Current : REAL
GET
                    Current := lCurrent;

                  
END_GET
END_PROPERTY

PROPERTY CurrentBMSChargeState : t_bms_charge_state
GET
                    CurrentBMSChargeState := lCurrentBMSChargeState;

                  
END_GET
END_PROPERTY

PROPERTY CurrentCoolantTemperature : REAL
GET
                    CurrentCoolantTemperature := lCurrentCoolantTemperature;
                  
END_GET
SET
                    lCurrentCoolantTemperature := CurrentCoolantTemperature;
                  
END_SET
END_PROPERTY

PROPERTY CurrentExceeding : REAL
GET
                    CurrentExceeding := lCurrentExceeding;
                  
END_GET
END_PROPERTY

PROPERTY CurrentLevel : t_percentage
GET
                    CurrentLevel := lCurrentLevel;
                  
END_GET
END_PROPERTY

PROPERTY CurrentState : t_bms_state
GET
                    CurrentState := lCurrentState;

                  
END_GET
END_PROPERTY

PROPERTY CurrentTMSState : t_tms_state
GET
                    CurrentTMSState := lCurrentTMSState;
                  
END_GET
SET
                    lCurrentTMSState := CurrentTMSState;
                  
END_SET
END_PROPERTY

PROPERTY DischargeCurrent : REAL
GET
                    DischargeCurrent := lDischargeCurrent;

                  
END_GET
END_PROPERTY

PROPERTY DischargeCurrentLimit : REAL
GET
                    DischargeCurrentLimit := lDischargeCurrentLimit;

                  
END_GET
END_PROPERTY

PROPERTY DischargeDerate : t_percentage
GET
                    DischargeDerate := lDischargeDerate;
                  
END_GET
END_PROPERTY

PROPERTY RequestedBMSChargeState : t_bms_charge_state
GET
                    RequestedBMSChargeState := lRequestedBMSChargeState;

                  
END_GET
SET
                    lRequestedBMSChargeState := RequestedBMSChargeState;
                  
END_SET
END_PROPERTY

PROPERTY RequestedCoolantTemperature : REAL
GET
                    RequestedCoolantTemperature := lRequestedCoolantTemperature;
                  
END_GET
END_PROPERTY

PROPERTY RequestedState : t_bms_state
GET
                    RequestedState := lRequestedState;

                  
END_GET
END_PROPERTY

PROPERTY RequestedTMSState : t_tms_state
GET
                    RequestedTMSState := lRequestedTMSState;
                  
END_GET
END_PROPERTY

PROPERTY SOC : t_percentage
GET
                    SOC := lSOC;
                  
END_GET
END_PROPERTY

PROPERTY TypeToken : t_medium_string
GET
                    TypeToken := 'BMS';
                  
END_GET
END_PROPERTY

PROPERTY Voltage : REAL
GET
                    Voltage := lVoltage;

                  
END_GET
END_PROPERTY

PROPERTY EnableBMS : UINT
SET
                    lEnableBMS.Value := EnableBMS;
                  
END_SET
END_PROPERTY

PROPERTY SOCMax : t_percentage
GET
                    SOCMax := lSOCMax;
                  
END_GET
END_PROPERTY

PROPERTY SOCMin : t_percentage
GET
                    SOCMin := lSOCMin;
                  
END_GET
END_PROPERTY
END_FUNCTION_BLOCK

FUNCTION_BLOCK BMSA EXTENDS BMS
  VAR
    lSOCA : t_percentage;
    lControllerBMSA : REFERENCE TO ControllerBMS;
  END_VAR

            ;
          

METHOD initialize
                  IF (NOT(__ISVALIDREF(lControllerBMSA))) THEN
	gCodeErrorHandler(pMessage:=CONCAT('null reference in ',lIdentity));
END_IF

SUPER^.initialize();

                
END_METHOD

METHOD operatorA
                  lCurrentState := lControllerBMSA.CurrentBMSState;

IF (lCurrentState=cBMSStateConnected) THEN
	lAvailability := 1.0;
ELSE
	lAvailability := 0.0;
END_IF

_operatorA();

SUPER^.operator();

lControllerBMSA.RequestedBMSState := lRequestedState;

                
END_METHOD

METHOD initializeBMS
  VAR_INPUT
    controllerBMSA : REFERENCE TO ControllerBMS;
  END_VAR
                  lControllerBMSA REF= controllerBMSA;

                
END_METHOD

METHOD operatorNull
                  lCurrentState := lRequestedState;

lAvailability := 0.0;

lSOC := 0.0;
lSOCMin := 0;
lSOCMax := 0;

lVoltage := 0.0;
lVoltageMin := 0;
lVoltageMax := 0;

lCurrent := 0.0;
lCurrentMin := 0;
lCurrentMax := 0;

_operatorNull();

SUPER^.operator();

lControllerBMSA.RequestedBMSState := cBMSStateDisconnected;

                
END_METHOD

METHOD _operatorA
                  lCurrentBMSChargeState := lControllerBMSA.CurrentBMSChargeState;
lRequestedTMSState := lControllerBMSA.RequestedTMSState;
lRequestedCoolantTemperature := lControllerBMSA.PackCoolantTemperatureTarget;
	
lBalancing := lControllerBMSA.Balancing;
	
lSOC := lControllerBMSA.PackSOC;
lSOCMin := lSOC;
lSOCMax := lSOC;

lVoltage := lControllerBMSA.PackVoltage;
lVoltageMin := lVoltage;
lVoltageMax := lVoltage;

lCurrent := lControllerBMSA.PackCurrent;
lCurrentMin := lCurrent;
lCurrentMax := lCurrent;

lChargeCurrent := lControllerBMSA.PackChargeCurrent;
lDischargeCurrent := lControllerBMSA.PackDischargeCurrent;

lChargeCurrentLimit := lControllerBMSA.PackChargeCurrentLimit;
lDischargeCurrentLimit := lControllerBMSA.PackDischargeCurrentLimit;
	
lChargingCurrentTarget := lControllerBMSA.PackChargingCurrentTarget;
lChargingVoltageTarget := lControllerBMSA.PackChargingVoltageTarget;

//lDischargePower := lControllerBMSA.DischargePower;
//lDischargeCumulativeEnergy := lControllerBMSA.DischargeCumulativeEnergy;
//lChargePower := lControllerBMSA.ChargePower;
//lChargeCumulativeEnergy := lControllerBMSA.ChargeCumulativeEnergy;


                
END_METHOD

METHOD operator
  VAR
    enableBMSA : BOOL;
  END_VAR
                  lSOCA := lControllerBMSA.PackSOC;

enableBMSA := UINT_TO_BOOL(lEnableBMS.Value AND 16#1);

IF (enableBMSA) THEN
	operatorA();
ELSE
	operatorNull();
END_IF

lControllerBMSA.RequestedBMSChargeState := lRequestedBMSChargeState;
lControllerBMSA.CurrentTMSState := lRequestedTMSState;

                
END_METHOD
END_FUNCTION_BLOCK

FUNCTION_BLOCK BMSAB EXTENDS BMS
  VAR_INPUT
    {attribute 'input_constant'}
    cVoltageMismatchThreshold : REAL := 0.5;
    {attribute 'input_constant'}
    cSOCMismatchThreshold : REAL := 0.05;
    {attribute 'input_constant'}
    cCurrentMismatchThreshold : REAL := 10.0;
  END_VAR
  VAR CONSTANT
    cSwitchingStatePeriod : t_time := TIME#1s500ms;
  END_VAR
  VAR
    lVRVoltageMismatchThreshold : ValueReferencePersistentReal;
    lVoltageMismatchThreshold : t_persistent_real;
    lVRSOCMismatchThreshold : ValueReferencePersistentReal;
    lSOCMismatchThreshold : t_persistent_real;
    lVRCurrentMismatchThreshold : ValueReferencePersistentReal;
    lCurrentMismatchThreshold : t_persistent_real;
    lVRDisableVoltageMismatchManagement : ValueReferencePersistentBool;
    lDisableVoltageMismatchManagement : t_persistent_bool;
    lVRAvailabilityFactor : ValueReferencePersistentReal;
    lAvailabilityFactor : t_persistent_real;
    lAlarmBMSSOCMismatch : ReportableAlarmEscalating;
    lAlarmBMSVoltageMismatch : ReportableAlarmEscalating;
    lAlarmBMSCurrentMismatch : ReportableAlarmEscalating;
    lAlarmTMSStateMismatch : ReportableAlarmEscalating;
    lAlarmBMSChargeStateMismatch : ReportableAlarmEscalating;
    lSOCA : t_percentage;
    lSOCB : t_percentage;
    lSOCMismatch : t_percentage;
    lSOCInbalance : t_percentage;
    lVoltageA : REAL;
    lVoltageB : REAL;
    lVoltageMismatch : REAL;
    lVoltageInbalance : t_percentage;
    lCurrentA : REAL;
    lCurrentB : REAL;
    lCurrentMismatch : REAL;
    lCurrentInbalance : t_percentage;
    lCurrentStateA : t_bms_state;
    lTargetStateA : t_bms_state;
    lRequestedStateA : t_bms_state;
    lCurrentStateB : t_bms_state;
    lTargetStateB : t_bms_state;
    lRequestedStateB : t_bms_state;
    lSwitchingStateTimer : t_timer;
    lControllerBMSA : REFERENCE TO ControllerBMS;
    lControllerBMSB : REFERENCE TO ControllerBMS;
  END_VAR

            ;
          

METHOD _operatorA
                  lCurrentBMSChargeState := lControllerBMSA.CurrentBMSChargeState;
lRequestedTMSState := lControllerBMSA.RequestedTMSState;
lRequestedCoolantTemperature := lControllerBMSA.PackCoolantTemperatureTarget;
	
lBalancing := lControllerBMSA.Balancing;
	
lSOC := lSOCA;
lSOCMin := lSOCA;
lSOCMax := lSOCA;
lVoltage := lVoltageA;
lVoltageMin := lVoltageA;
lVoltageMax := lVoltageA;

lCurrent := lControllerBMSA.PackCurrent;
lChargeCurrent := lControllerBMSA.PackChargeCurrent;
lDischargeCurrent := lControllerBMSA.PackDischargeCurrent;

lChargeCurrentLimit := lControllerBMSA.PackChargeCurrentLimit;
lDischargeCurrentLimit := lControllerBMSA.PackDischargeCurrentLimit;
	
lChargingCurrentTarget := lControllerBMSA.PackChargingCurrentTarget;
lChargingVoltageTarget := lControllerBMSA.PackChargingVoltageTarget;

//lDischargePower := lControllerBMSA.DischargePower;
//lDischargeCumulativeEnergy := lControllerBMSA.DischargeCumulativeEnergy;
//lChargePower := lControllerBMSA.ChargePower;
//lChargeCumulativeEnergy := lControllerBMSA.ChargeCumulativeEnergy;


                
END_METHOD

METHOD _operatorAB
                  lCurrentBMSChargeState := MIN(lControllerBMSA.CurrentBMSChargeState,
	lControllerBMSB.CurrentBMSChargeState);

IF (lControllerBMSA.CurrentBMSChargeState<>lControllerBMSB.CurrentBMSChargeState) THEN
	lAlarmBMSChargeStateMismatch.trigger(FALSE); // foobar any further action
END_IF

resolveRequestedTMSState();

lBalancing := ((lControllerBMSA.Balancing) OR
	(lControllerBMSB.Balancing));
	
lSOC := MIN(lSOCA,lSOCB);
lSOCMin := MIN(lSOCA,lSOCB);
lSOCMax := MAX(lSOCA,lSOCB);

lVoltage := (lVoltageA + lVoltageB)/2.0;
lVoltageMin := MIN(lVoltageA,lVoltageB);
lVoltageMax := MAX(lVoltageA,lVoltageB);

lCurrent := lCurrentA + lCurrentB;
lCurrentMin := MIN(lCurrentA,lCurrentB);
lCurrentMax := MAX(lCurrentA,lCurrentB);

IF (lCurrentMismatch>lCurrentMismatchThreshold.Value) THEN
	lAlarmBMSCurrentMismatch.trigger(FALSE);
END_IF

lChargeCurrent := lControllerBMSA.PackChargeCurrent + lControllerBMSB.PackChargeCurrent;
lDischargeCurrent := lControllerBMSA.PackDischargeCurrent + lControllerBMSB.PackDischargeCurrent;

lChargeCurrentLimit := lControllerBMSA.PackChargeCurrentLimit + lControllerBMSB.PackChargeCurrentLimit; // foobar how to test charge/discharge modulation
lDischargeCurrentLimit := lControllerBMSA.PackDischargeCurrentLimit + lControllerBMSB.PackDischargeCurrentLimit;
	
lChargingCurrentTarget := lControllerBMSA.PackChargingCurrentTarget + lControllerBMSB.PackChargingCurrentTarget;
lChargingVoltageTarget := MIN(lControllerBMSA.PackChargingVoltageTarget,lControllerBMSB.PackChargingVoltageTarget);

//foostrip lDischargePower := lControllerBMSA.DischargePower + lControllerBMSB.DischargePower;
//lDischargeCumulativeEnergy := lControllerBMSA.DischargeCumulativeEnergy + lControllerBMSB.DischargeCumulativeEnergy;
//lChargePower := lControllerBMSA.ChargePower + lControllerBMSB.ChargePower;
//lChargeCumulativeEnergy := lControllerBMSA.ChargeCumulativeEnergy + lControllerBMSB.ChargeCumulativeEnergy;




                
END_METHOD

METHOD _operatorB
                  lCurrentBMSChargeState := lControllerBMSB.CurrentBMSChargeState;
lRequestedTMSState := lControllerBMSB.RequestedTMSState;
lRequestedCoolantTemperature := lControllerBMSB.PackCoolantTemperatureTarget;
	
lBalancing := lControllerBMSB.Balancing;
	
lSOC := lSOCB;
lSOCMin := lSOCB;
lSOCMax := lSOCB;
lVoltage := lVoltageB;
lVoltageMin := lVoltageB;
lVoltageMax := lVoltageB;

lCurrent := lControllerBMSB.PackCurrent;
lChargeCurrent := lControllerBMSB.PackChargeCurrent;
lDischargeCurrent := lControllerBMSB.PackDischargeCurrent;

lChargeCurrentLimit := lControllerBMSB.PackChargeCurrentLimit;
lDischargeCurrentLimit := lControllerBMSB.PackDischargeCurrentLimit;
	
lChargingCurrentTarget := lControllerBMSB.PackChargingCurrentTarget;
lChargingVoltageTarget := lControllerBMSB.PackChargingVoltageTarget;

//lDischargePower := lControllerBMSB.DischargePower;
//lDischargeCumulativeEnergy := lControllerBMSB.DischargeCumulativeEnergy;
//lChargePower := lControllerBMSB.ChargePower;
//lChargeCumulativeEnergy := lControllerBMSB.ChargeCumulativeEnergy;


                
END_METHOD

METHOD initialize
                  IF ((NOT(__ISVALIDREF(lControllerBMSA))) OR
	(NOT(__ISVALIDREF(lControllerBMSB)))) THEN
	gCodeErrorHandler(pMessage:=CONCAT('null reference in ',lIdentity));
END_IF

lVRVoltageMismatchThreshold.initializeValueReference(lVoltageMismatchThreshold,NopSelf,'VoltageMismatch','Maximum allowable difference between BMS voltages','',cValueStyleParameter);
lVoltageMismatchThreshold.Identifier := t_persistent_id.cPersistentID_VoltageMismatchThreshold;
lVoltageMismatchThreshold.initialize();
IF (lVoltageMismatchThreshold.Value=0.0) THEN
	lVoltageMismatchThreshold.Value := cVoltageMismatchThreshold;
END_IF

lVRSOCMismatchThreshold.initializeValueReference(lSOCMismatchThreshold,NopSelf,'SOCMismatch','Maximum allowable difference between BMS SOCs','',cValueStyleParameter);
lSOCMismatchThreshold.Identifier := t_persistent_id.cPersistentID_SOCMismatchThreshold;
lSOCMismatchThreshold.initialize();
IF (lSOCMismatchThreshold.Value=0.0) THEN
	lSOCMismatchThreshold.Value := cSOCMismatchThreshold;
END_IF

lVRCurrentMismatchThreshold.initializeValueReference(lCurrentMismatchThreshold,NopSelf,'CurrentMismatch','Maximum allowable difference between BMS currents','',cValueStyleParameter);
lCurrentMismatchThreshold.Identifier := t_persistent_id.cPersistentID_CurrentMismatchThreshold;
lCurrentMismatchThreshold.initialize();
IF (lCurrentMismatchThreshold.Value=0.0) THEN
	lCurrentMismatchThreshold.Value := cCurrentMismatchThreshold;
END_IF

lVRDisableVoltageMismatchManagement.initializeValueReference(lDisableVoltageMismatchManagement,NopSelf,'DsblVoltMisMgmt','Disable voltage mismatch checking between BMS voltages','',cValueStyleParameter);
lDisableVoltageMismatchManagement.Identifier := t_persistent_id.cPersistentID_VoltageMismatchManagement;
lDisableVoltageMismatchManagement.initialize();

lVRAvailabilityFactor.initializeValueReference(lAvailabilityFactor,NopSelf,'AvailFactor','Factor used to calculate BMS availability','',cValueStyleParameter);
lAvailabilityFactor.Identifier := t_persistent_id.cPersistentID_BMSAvailabilityFactor;
lAvailabilityFactor.initialize();

lAlarmTMSStateMismatch.initializeState(NopSelf,'',cACTMSStateMismatch);
lAlarmTMSStateMismatch.Life := 10;
lAlarmTMSStateMismatch.InitialSeverity := cSeverityNone;
lAlarmTMSStateMismatch.SeverityWarningTimeout := T#30S;
lAlarmTMSStateMismatch.SeverityErrorTimeout := T#200S;
lAlarmTMSStateMismatch.SeverityCriticalTimeout := T#300S;

lAlarmBMSChargeStateMismatch.initializeState(NopSelf,'',cACBMSChargeStateMismatch);
lAlarmBMSChargeStateMismatch.Life := 10;
lAlarmBMSChargeStateMismatch.InitialSeverity := cSeverityNone;
lAlarmBMSChargeStateMismatch.SeverityWarningTimeout := T#1S;
lAlarmBMSChargeStateMismatch.SeverityErrorTimeout := T#2S;
lAlarmBMSChargeStateMismatch.SeverityCriticalTimeout := T#5S;

lAlarmBMSVoltageMismatch.initializeState(NopSelf,'',cACBMSVoltageMismatch);
lAlarmBMSVoltageMismatch.Life := 10;
lAlarmBMSVoltageMismatch.InitialSeverity := cSeverityNone;
lAlarmBMSVoltageMismatch.SeverityWarningTimeout := T#1S;
lAlarmBMSVoltageMismatch.SeverityErrorTimeout := T#2S;
lAlarmBMSVoltageMismatch.SeverityCriticalTimeout := T#5S;

lAlarmBMSSOCMismatch.initializeState(NopSelf,'',cACBMSSOCMismatch);
lAlarmBMSSOCMismatch.Life := 10;
lAlarmBMSSOCMismatch.InitialSeverity := cSeverityNone;
lAlarmBMSSOCMismatch.SeverityWarningTimeout := T#1S;
lAlarmBMSSOCMismatch.SeverityErrorTimeout := T#2S;
lAlarmBMSSOCMismatch.SeverityCriticalTimeout := T#5S;

lAlarmBMSCurrentMismatch.initializeState(NopSelf,'',cACBMSCurrentMismatch);
lAlarmBMSCurrentMismatch.Life := 10;
lAlarmBMSCurrentMismatch.InitialSeverity := cSeverityNone;
lAlarmBMSCurrentMismatch.SeverityWarningTimeout := T#1S;
lAlarmBMSCurrentMismatch.SeverityErrorTimeout := T#2S;
lAlarmBMSCurrentMismatch.SeverityCriticalTimeout := T#5S;

SUPER^.initialize();

lSwitchingStateTimer.Enable := TRUE;
lSwitchingStateTimer.Period := cSwitchingStatePeriod;
lSwitchingStateTimer.initialize();

                
END_METHOD

METHOD operator
  VAR
    enableBMSA : BOOL;
    enableBMSB : BOOL;
  END_VAR
                  lCurrentStateA := lControllerBMSA.CurrentBMSState;
lCurrentStateB := lControllerBMSB.CurrentBMSState;

lSOCA := lControllerBMSA.PackSOC;
lSOCB := lControllerBMSB.PackSOC;
lSOCMismatch := ABS(lSOCA - lSOCB);
lSOCInbalance := ABS(lSOCA/lSOCB);

IF (lSOCMismatch>lSOCMismatchThreshold.Value) THEN
	lAlarmBMSSOCMismatch.trigger(FALSE);
END_IF

lVoltageA := lControllerBMSA.PackVoltage;
lVoltageB := lControllerBMSB.PackVoltage;
lVoltageMismatch := ABS(lVoltageA-lVoltageB);
lVoltageInbalance := ABS(lVoltageA/lVoltageB);

IF (lVoltageMismatch>lVoltageMismatchThreshold.Value) THEN
	lAlarmBMSVoltageMismatch.trigger(FALSE);
END_IF

lCurrentA := lControllerBMSA.PackCurrent;
lCurrentB := lControllerBMSB.PackCurrent;
lCurrentMismatch := ABS(lCurrentA-lCurrentB);
lCurrentInbalance := ABS(lCurrentA/lCurrentB);

enableBMSA := UINT_TO_BOOL(lEnableBMS.Value AND 16#1);
enableBMSB := UINT_TO_BOOL(lEnableBMS.Value AND 16#2);

IF ((enableBMSA) AND (NOT(enableBMSB))) THEN
	operatorA();
ELSIF ((enableBMSB) AND (NOT(enableBMSA))) THEN
	operatorB();
ELSIF ((enableBMSB) AND (enableBMSA)) THEN
	operatorAB();
ELSE
	operatorNull();
END_IF

processRequestedBMSState();

lControllerBMSA.RequestedBMSChargeState := lRequestedBMSChargeState;
lControllerBMSB.RequestedBMSChargeState := lRequestedBMSChargeState;

lControllerBMSA.CurrentTMSState := lRequestedTMSState;
lControllerBMSB.CurrentTMSState := lRequestedTMSState;

                
END_METHOD

METHOD operatorA
                  lCurrentState := lControllerBMSA.CurrentBMSState;

IF (lCurrentState=cBMSStateConnected) THEN
	lAvailability := lAvailabilityFactor.Value;
ELSE
	lAvailability := 0.0;
END_IF

_operatorA();

SUPER^.operator();

lTargetStateA := lRequestedState;
lTargetStateB := cBMSStateDisconnected;

                
END_METHOD

METHOD operatorAB
                  lCurrentState := MAX(lCurrentStateA,lCurrentStateB);

lAvailability := 0.0;
IF (lCurrentStateA=cBMSStateConnected) THEN
	lAvailability := MIN(lAvailability + lAvailabilityFactor.Value,1.0);
END_IF
IF (lCurrentStateB=cBMSStateConnected) THEN
	lAvailability := MIN(lAvailability + lAvailabilityFactor.Value,1.0);
END_IF

IF ((lCurrentStateA=cBMSStateConnected) AND
	(lCurrentStateB<>cBMSStateConnected)) THEN
	_operatorA();

ELSIF ((lCurrentStateB=cBMSStateConnected) AND
	(lCurrentStateA<>cBMSStateConnected)) THEN
	_operatorB();

ELSIF ((lCurrentStateB=cBMSStateConnected) AND
	(lCurrentStateA=cBMSStateConnected)) THEN
	_operatorAB();

ELSE
	lSOC := (lSOCA + lSOCB)/2.0;
	lSOCMin := MIN(lSOCA,lSOCB);
	lSOCMax := MAX(lSOCA,lSOCB);
	
	lVoltage := (lVoltageA + lVoltageB)/2.0;
	lVoltageMin := MIN(lVoltageA,lVoltageB);
	lVoltageMax := MAX(lVoltageA,lVoltageB);
	
	lCurrent := lCurrentA + lCurrentB;
	lCurrentMin := MIN(lCurrentA,lCurrentB);
	lCurrentMax := MAX(lCurrentA,lCurrentB);
	
	_operatorNull();
END_IF

SUPER^.operator();

resolveRequestedBMSState();

                
END_METHOD

METHOD operatorB
                  lCurrentState := lControllerBMSB.CurrentBMSState;

IF (lCurrentState=cBMSStateConnected) THEN
	lAvailability := lAvailabilityFactor.Value;
ELSE
	lAvailability := 0.0;
END_IF

_operatorB();

SUPER^.operator();

lTargetStateA := cBMSStateDisconnected;
lTargetStateB := lRequestedState;

                
END_METHOD

METHOD resolveRequestedTMSState
                  IF (lControllerBMSA.RequestedTMSState=lControllerBMSB.RequestedTMSState) THEN
	lRequestedTMSState := lControllerBMSA.RequestedTMSState;
	lRequestedCoolantTemperature := MIN(lControllerBMSA.PackCoolantTemperatureTarget,lControllerBMSB.PackCoolantTemperatureTarget);

	IF (lRequestedTMSState=cTMSStateHeating) THEN
		lRequestedCoolantTemperature := MAX(lControllerBMSA.PackCoolantTemperatureTarget,lControllerBMSB.PackCoolantTemperatureTarget);
	END_IF
	
	RETURN;
END_IF

IF (lControllerBMSA.RequestedTMSState<>lControllerBMSB.RequestedTMSState) THEN
	lAlarmTMSStateMismatch.trigger(FALSE); // foobar any further action
END_IF

IF ((lControllerBMSA.RequestedTMSState=cTMSStateCooling) OR
	(lControllerBMSB.RequestedTMSState=cTMSStateCooling)) THEN
	lRequestedTMSState := cTMSStateCooling;
	lRequestedCoolantTemperature := MIN(lControllerBMSA.PackCoolantTemperatureTarget,lControllerBMSB.PackCoolantTemperatureTarget);
	RETURN;
END_IF

IF ((lControllerBMSA.RequestedTMSState=cTMSStateHeating) OR
	(lControllerBMSB.RequestedTMSState=cTMSStateHeating)) THEN
	lRequestedTMSState := cTMSStateHeating;
	lRequestedCoolantTemperature := MAX(lControllerBMSA.PackCoolantTemperatureTarget,lControllerBMSB.PackCoolantTemperatureTarget);
	RETURN;
END_IF

lRequestedCoolantTemperature := MIN(lControllerBMSA.PackCoolantTemperatureTarget,lControllerBMSB.PackCoolantTemperatureTarget);

IF ((lControllerBMSA.RequestedTMSState=cTMSStateCirculation) OR
	(lControllerBMSB.RequestedTMSState=cTMSStateCirculation)) THEN
	lRequestedTMSState := cTMSStateCirculation;
	RETURN;
END_IF

lRequestedTMSState := cTMSStateShutdown;


                
END_METHOD

METHOD initializeBMS
  VAR_INPUT
    controllerBMSA : REFERENCE TO ControllerBMS;
    controllerBMSB : REFERENCE TO ControllerBMS;
  END_VAR
                  lControllerBMSA REF= controllerBMSA;
lControllerBMSB REF= controllerBMSB;
                
END_METHOD

METHOD operatorNull
                  lCurrentState := lRequestedState;

lAvailability := 0.0;
lSOC := 0.0;
lSOCMin := 0;
lSOCMax := 0;
lVoltage := 0.0;
lVoltageMin := 0;
lVoltageMax := 0;


_operatorNull();

SUPER^.operator();

lTargetStateA := cBMSStateDisconnected;
lTargetStateB := cBMSStateDisconnected;

                
END_METHOD

METHOD resolveRequestedBMSState
                  IF (lRequestedState<>cBMSStateConnected) THEN
	lTargetStateA := lRequestedState;
	lTargetStateB := lRequestedState;
	
	RETURN;
END_IF

IF ((gSystemServices.SystemState.State<=cSystemStatePreparing) AND
	(NOT(lDisableVoltageMismatchManagement.Value))) THEN

	IF (lVoltageA>(lVoltageB+lVoltageMismatchThreshold.Value)) THEN
		IF (gSystemServices.SystemState.ChargingEnabled) THEN
			lTargetStateA := cBMSStateDisconnected;
			lTargetStateB := cBMSStateConnected;		
		ELSE
			lTargetStateA := cBMSStateConnected;
			lTargetStateB := cBMSStateDisconnected;
		END_IF
		
		RETURN;
	END_IF
	
	IF (lVoltageB>(lVoltageA+lVoltageMismatchThreshold.Value)) THEN
		IF (gSystemServices.SystemState.ChargingEnabled) THEN
			lTargetStateA := cBMSStateConnected;
			lTargetStateB := cBMSStateDisconnected;
		ELSE
			lTargetStateA := cBMSStateDisconnected;
			lTargetStateB := cBMSStateConnected;
		END_IF

		RETURN;
	END_IF
END_IF

IF (lCurrentStateA<cBMSStateDisconnected) THEN
	lTargetStateA := cBMSStateDisconnected;
ELSE
	lTargetStateA := cBMSStateConnected;
END_IF

IF (lCurrentStateB<cBMSStateDisconnected) THEN
	lTargetStateB := cBMSStateDisconnected;
ELSE
	lTargetStateB := cBMSStateConnected;
END_IF

                
END_METHOD

METHOD processRequestedBMSState
                  IF ((lTargetStateA=lCurrentStateA) AND
	(lTargetStateB=lCurrentStateB)) THEN
	lSwitchingStateTimer.reset();	
END_IF
lSwitchingStateTimer.operator();

IF (lTargetStateA<>cBMSStateConnected) THEN
	lRequestedStateA := lTargetStateA;
ELSE
	IF (lSwitchingStateTimer.Expired) THEN
		lRequestedStateA := lTargetStateA;
	ELSE
		lRequestedStateA := lCurrentStateA;
	END_IF
END_IF

IF (lTargetStateB<>cBMSStateConnected) THEN
	lRequestedStateB := lTargetStateB;
ELSE
	IF (lSwitchingStateTimer.Expired) THEN
		lRequestedStateB := lTargetStateB;
	ELSE
		lRequestedStateB := lCurrentStateB;
	END_IF
END_IF

lControllerBMSA.RequestedBMSState := lRequestedStateA;	
lControllerBMSB.RequestedBMSState := lRequestedStateB;	

                
END_METHOD

PROPERTY TypeToken : t_medium_string
GET
                    TypeToken := 'BMSAB';
                  
END_GET
END_PROPERTY
END_FUNCTION_BLOCK

FUNCTION_BLOCK TMS EXTENDS OperationalParticleSet
  VAR CONSTANT
    cCoolantTempHotInitialCutbackThreshold : REAL := 45;
    cCoolantTempHotCutoutThreshold : REAL := 35;
    cCoolantTempColdInitialCutbackThreshold : REAL := 5;
    cCoolantTempColdCutoutThreshold : REAL := -10;
    cCoolantTempCriticalUpperThreshold : REAL := 22;  (* foobar persistent? adaptive? *)
    cCoolantTempCriticalUpperHysteresis : REAL := 2;
    cCoolantTempCriticalLowerThreshold : REAL := 4;
    cCoolantTempCriticalLowerHysteresis : REAL := 2;
    cSecondaryRequiredAvailabilityHeatingCooling : t_percentage := 1.0;
    cSecondaryRequiredAvailabilityPump : t_percentage := 0.3;
  END_VAR
  VAR
    lAlarmCoolantReservoirLow : ReportableAlarmEscalating;
    lAlarmSecondaryPowerFailHeatingCooling : ReportableAlarmEscalating;
    lAlarmSecondaryPowerFailPump : ReportableAlarmEscalating;
    lDiagnosticTMSCooling : ReportableDiagnostic;
    lDiagnosticTMSHeating : ReportableDiagnostic;
    lDiagnosticBMSTMSCooling : ReportableDiagnostic;
    lDiagnosticBMSTMSHeating : ReportableDiagnostic;
    lDiagnosticBMSTMSNoCirculation : ReportableDiagnostic;
    lAlarmCoolantHeating : ReportableAlarmEscalating;
    lAlarmCoolantChilling : ReportableAlarmEscalating;
    lAlarmCoolantTempHotCutback : CutbackInterlock;
    lAlarmCoolantTempColdCutback : CutbackInterlock;
    lVROverrideControl : ValueReferenceBool;
    lOverrideControl : BOOL := FALSE;
    lCurrentCoolantTemperature : ValueObjectRealScaledOffsetInputReferenceDINT;
    lCoolantReservoir : ValueObjectBoolInputReferenceDINTAsBool;
    lCoolantTemperatureCriticalUpper : ValueObjectBoolInputRealThreshold;
    lCoolantTemperatureCriticalLower : ValueObjectBoolInputRealThreshold;
    lCoolantPump : ValueObjectBoolOutputReferenceDINTAsBool;
    lCoolantHeating : ValueObjectBoolCheckReferenceDINTOutputReferenceDINT;
    lCoolantChilling : ValueObjectBoolOutputReferenceDINTAsBool;
    lRequestedState : ValueObjectEnumType;
    lCurrentState : ValueObjectEnumType;
    lRequestedCoolantTemperature : REAL;
  END_VAR

            ;
          

METHOD initialize
                  lAlarmCoolantReservoirLow.initializeState(NopSelf,'',cACCoolantReservoir);
lAlarmCoolantReservoirLow.Life := 10;
lAlarmCoolantReservoirLow.InitialSeverity := cSeverityNone;
lAlarmCoolantReservoirLow.SeverityWarningTimeout := T#1S;
lAlarmCoolantReservoirLow.SeverityErrorTimeout := T#2S;
lAlarmCoolantReservoirLow.SeverityCriticalTimeout := T#2H;

lAlarmSecondaryPowerFailHeatingCooling.InitialSeverity := cSeverityWarning;
lAlarmSecondaryPowerFailHeatingCooling.SeverityWarningTimeout := T#1S;
lAlarmSecondaryPowerFailHeatingCooling.initializeState(NopSelf,'',cACCoolantSecondaryPowerFailHeatingCooling);
lAlarmSecondaryPowerFailHeatingCooling.Life := 10;
lAlarmSecondaryPowerFailHeatingCooling.SeverityErrorTimeout := T#2S;
lAlarmSecondaryPowerFailHeatingCooling.SeverityCriticalTimeout := T#5S;

lAlarmSecondaryPowerFailPump.initializeState(NopSelf,'',cACCoolantSecondaryPowerFailPump);
lAlarmSecondaryPowerFailPump.Life := 10;
lAlarmSecondaryPowerFailPump.InitialSeverity := cSeverityWarning;
lAlarmSecondaryPowerFailPump.SeverityWarningTimeout := T#1S;
lAlarmSecondaryPowerFailPump.SeverityErrorTimeout := T#2S;
lAlarmSecondaryPowerFailPump.SeverityCriticalTimeout := T#5S;
	
lDiagnosticTMSCooling.initializeState(NopSelf,'',cDCTMSCooling);
lDiagnosticTMSHeating.initializeState(NopSelf,'',cDCTMSHeating);
lDiagnosticBMSTMSCooling.initializeState(NopSelf,'',cDCBMSTMSCooling);
lDiagnosticBMSTMSHeating.initializeState(NopSelf,'',cDCBMSTMSHeating);
lDiagnosticBMSTMSNoCirculation.initializeState(NopSelf,'',cDCBMSTMSNoCirculation);
	
lAlarmCoolantHeating.initializeState(NopSelf,'',cACCoolantHeating);
lAlarmCoolantHeating.InitialSeverity := cSeverityNone;
lAlarmCoolantHeating.SeverityWarningTimeout := T#1S;
lAlarmCoolantHeating.SeverityErrorTimeout := T#2S;
lAlarmCoolantHeating.SeverityCriticalTimeout := T#5S;

lAlarmCoolantChilling.initializeState(NopSelf,'',cACCoolantChilling);
lAlarmCoolantChilling.InitialSeverity := cSeverityNone;
lAlarmCoolantChilling.SeverityWarningTimeout := T#1S;
lAlarmCoolantChilling.SeverityErrorTimeout := T#2S;
lAlarmCoolantChilling.SeverityCriticalTimeout := T#5S;

lAlarmCoolantTempHotCutback.initializeState(NopSelf,'',cACCoolantTempHotCutback);
lAlarmCoolantTempHotCutback.Qualifier := cChargeQualifierBoth;
lAlarmCoolantTempHotCutback.InitialCutbackThreshold :=cCoolantTempHotInitialCutbackThreshold;
lAlarmCoolantTempHotCutback.CutoutThreshold := cCoolantTempHotCutoutThreshold;
lAlarmCoolantTempHotCutback.registerServer(gSystemPrimary.Travel.ChargeInterlock);
lAlarmCoolantTempHotCutback.registerServer(gSystemPrimary.Lift.ChargeInterlock);

lAlarmCoolantTempColdCutback.initializeState(NopSelf,'',cACCoolantTempColdCutback);
lAlarmCoolantTempColdCutback.Qualifier := cChargeQualifierBoth;
lAlarmCoolantTempColdCutback.InitialCutbackThreshold :=cCoolantTempColdInitialCutbackThreshold;
lAlarmCoolantTempColdCutback.CutoutThreshold := cCoolantTempColdCutoutThreshold;
lAlarmCoolantTempColdCutback.registerServer(gSystemPrimary.Travel.ChargeInterlock);
lAlarmCoolantTempColdCutback.registerServer(gSystemPrimary.Lift.ChargeInterlock);

lVROverrideControl.initializeValueReference(lOverrideControl,NopSelf,'OvrdControl','Override TMS automatic control','',cValueStyleParameter);

lRequestedState.EnumType := cEnumTypeTMSState;
lRequestedState.initializeValueObject(NopSelf,'ReqState','Requested TMS state','',cValueStyleConfigurable);

lCurrentState.EnumType := cEnumTypeTMSState;
lCurrentState.initializeValueObjectOp(OpSelf,'CurrState','Current TMS state','',cValueStyleConfigurable);

lCoolantReservoir.initializeValueObjectOp(OpSelf,'ClntReservoir','Battery coolant reservoir state','',cValueStyleConfigurable);

lCurrentCoolantTemperature.Offset := -22.522;
lCurrentCoolantTemperature.Scaling := 0.0314;
lCurrentCoolantTemperature.initializeValueObjectOp(OpSelf,'ClntTemp','Battery coolant temperature','celcius',cValueStyleConfigurable);

lCoolantTemperatureCriticalUpper.Threshold := cCoolantTempCriticalUpperThreshold;
lCoolantTemperatureCriticalUpper.Hysteresis := cCoolantTempCriticalUpperHysteresis;
lCoolantTemperatureCriticalUpper.BelowIsOn := FALSE;
lCoolantTemperatureCriticalUpper.initializeValueObject(NopSelf,'ClntTempHot','Battery coolant temperature is hot','',cValueStyleConfigurable);

lCoolantTemperatureCriticalLower.Threshold := cCoolantTempCriticalLowerThreshold;
lCoolantTemperatureCriticalLower.Hysteresis := cCoolantTempCriticalLowerHysteresis;
lCoolantTemperatureCriticalLower.BelowIsOn := TRUE;
lCoolantTemperatureCriticalLower.initializeValueObject(NopSelf,'ClntTempCold','Battery coolant temperature is cold','',cValueStyleConfigurable);

lCoolantPump.initializeValueObjectOp(OpSelf,'Pump','Battery coolant pump is running','',cValueStyleConfigurable);

lCoolantHeating.CheckEnable := TRUE;
lCoolantHeating.CheckCritical := TRUE;
lCoolantHeating.CheckPeriod := cRelayCoilTimeout;
lCoolantHeating.initializeValueObjectOp(OpSelf,'Heating','Battery coolant heater is running','',cValueStyleConfigurable);

lCoolantChilling.initializeValueObjectOp(OpSelf,'Chilling','Battery coolant chiller is running','',cValueStyleConfigurable);

SUPER^.initialize();
SubSystem := cSubsystemBattery;

lRequestedState.Value := cTMSStateShutdown;
lCurrentState.Value := cTMSStateShutdown;

                
END_METHOD

METHOD operator
                  lRequestedCoolantTemperature := gSystemPrimary.BMS.RequestedCoolantTemperature; //foobar ignored

lRequestedState.Value := gSystemPrimary.BMS.RequestedTMSState;
lRequestedState.operator();

CASE RequestedState OF
	cTMSStateShutdown:
		lCoolantPump.off();
		lCoolantHeating.off();
		lCoolantChilling.off();

		IF (gSystemPrimary.SystemState.State=cSystemStateOperational) THEN
			lDiagnosticBMSTMSNoCirculation.trigger(FALSE);
		END_IF

	cTMSStateCooling:
		lCoolantPump.on();
		lCoolantHeating.off();
		lCoolantChilling.on();
		lDiagnosticBMSTMSCooling.trigger(FALSE);

	cTMSStateHeating:
		lCoolantPump.on();
		lCoolantHeating.on();
		lCoolantChilling.off();
		lDiagnosticBMSTMSHeating.trigger(FALSE);
		
	cTMSStateCirculation:
		lCoolantPump.on();
		lCoolantHeating.off();
		lCoolantChilling.off();
END_CASE
lCurrentState.Value := RequestedState;

// following are TMS-independent actions that override instructions from the rest of the system

lCoolantTemperatureCriticalUpper.Input := lCurrentCoolantTemperature.Value;
IF (lCoolantTemperatureCriticalUpper.Value) THEN
	lCoolantPump.on();
	lCoolantHeating.off();
	lCoolantChilling.on();
	lDiagnosticTMSCooling.trigger(FALSE);

	lCurrentState.Value := cTMSStateCooling;
END_IF

lCoolantTemperatureCriticalLower.Input := lCurrentCoolantTemperature.Value;
IF (lCoolantTemperatureCriticalLower.Value) THEN
	lCoolantPump.on();
	lCoolantHeating.on();
	lCoolantChilling.off();
	lDiagnosticTMSHeating.trigger(FALSE);
	
	lCurrentState.Value := cTMSStateHeating;
END_IF

IF (gSystemPrimary.SystemState.State>=cSystemStatePreparing) THEN
	lCoolantPump.on();
END_IF

// checks on TMS-independent actions

IF ((lOverrideControl) OR
	(gSystemPrimary.BMS.Availability=0)) THEN
	lCurrentState.Value := cTMSStateShutdown;	

	lCoolantPump.off();
	lCoolantHeating.off();
	lCoolantChilling.off();
END_IF

IF (((lCoolantHeating.Value) OR (lCoolantChilling.Value)) AND
	(gSystemPrimary.lSecondaryPowerSupply.Availability<cSecondaryRequiredAvailabilityHeatingCooling)) THEN	
	lAlarmSecondaryPowerFailHeatingCooling.trigger(FALSE);

	lCoolantHeating.off();
	lCoolantChilling.off();	
END_IF

IF ((lCoolantPump.Value) AND
	(gSystemPrimary.lSecondaryPowerSupply.Availability<cSecondaryRequiredAvailabilityPump)) THEN
	lAlarmSecondaryPowerFailPump.trigger(FALSE);

	lCoolantPump.off();
END_IF

SUPER^.operator();

gSystemPrimary.BMS.CurrentTMSState := CurrentState;
gSystemPrimary.BMS.CurrentCoolantTemperature := lCurrentCoolantTemperature.Value;

lAlarmCoolantTempColdCutback.Value := lCurrentCoolantTemperature.Value;
lAlarmCoolantTempColdCutback.test(FALSE);

lAlarmCoolantTempHotCutback.Value := lCurrentCoolantTemperature.Value;
lAlarmCoolantTempHotCutback.test(FALSE);

IF ((gSystemPrimary.lSensorSupply.OK) AND
	(NOT(lCoolantReservoir.Value))) THEN
	lAlarmCoolantReservoirLow.trigger(FALSE);
END_IF

IF (lCoolantHeating.lError) THEN
	IF (RequestedState=cTMSStateHeating) THEN
		lCurrentState.Value := cTMSStateCirculation;
	END_IF
	
	lAlarmCoolantHeating.trigger(FALSE);
END_IF

IF (FALSE) THEN // foobar, a different way of checking chilling function is required
	IF (RequestedState=cTMSStateCooling) THEN
		lCurrentState.Value := cTMSStateCirculation;
	END_IF

	lAlarmCoolantChilling.trigger(FALSE);
END_IF

                
END_METHOD

METHOD initializeTMS
  VAR_INPUT
    inputCoolantTemperature : REFERENCE TO DINT;
    inputCoolantReservoir : REFERENCE TO DINT;
    outputCoolantPump : REFERENCE TO DINT;
    outputCoolantHeating : REFERENCE TO DINT;
    inputCheckCoolantHeating : REFERENCE TO DINT;
    outputCoolantChillerA : REFERENCE TO DINT;
  END_VAR
                  lCurrentCoolantTemperature.InputReference REF= inputCoolantTemperature;
lCoolantReservoir.InputReference REF= inputCoolantReservoir;

lCoolantPump.OutputReference REF= outputCoolantPump;
lCoolantHeating.OutputReference REF= outputCoolantHeating;
lCoolantHeating.CheckReference REF= inputCheckCoolantHeating;
lCoolantChilling.OutputReference REF= outputCoolantChillerA;

	
	
	
	
	
	
	
                
END_METHOD

PROPERTY CoolantChillingObject : REFERENCE TO ValueObjectBool
GET
                    CoolantChillingObject REF= lCoolantChilling;

                  
END_GET
END_PROPERTY

PROPERTY CoolantHeatingObject : REFERENCE TO ValueObjectBool
GET
                    CoolantHeatingObject REF= lCoolantHeating;

                  
END_GET
END_PROPERTY

PROPERTY CoolantPumpObject : REFERENCE TO ValueObjectBool
GET
                    CoolantPumpObject REF= lCoolantPump;

                  
END_GET
END_PROPERTY

PROPERTY CoolantReservoir : BOOL
GET
                    CoolantReservoir := lCoolantReservoir.Value;
                  
END_GET
END_PROPERTY

PROPERTY CoolantTemperatureCritical : BOOL
GET
                    CoolantTemperatureCritical := lCoolantTemperatureCriticalUpper.Value;
                  
END_GET
END_PROPERTY

PROPERTY CurrentCoolantTemperature : REAL
GET
                    CurrentCoolantTemperature := lCurrentCoolantTemperature.Value;
                  
END_GET
END_PROPERTY

PROPERTY CurrentCoolantTemperatureObject : REFERENCE TO ValueObjectReal
GET
                    CurrentCoolantTemperatureObject REF= lCurrentCoolantTemperature;

                  
END_GET
END_PROPERTY

PROPERTY CurrentState : t_tms_state
GET
                    CurrentState := lCurrentState.Value;
                  
END_GET
END_PROPERTY

PROPERTY RequestedCoolantTemperature : REAL
GET
                    
                  
END_GET
END_PROPERTY

PROPERTY RequestedState : t_tms_state
GET
                    RequestedState := lRequestedState.Value;
                  
END_GET
END_PROPERTY

PROPERTY TypeToken : t_medium_string
GET
                    TypeToken := 'TMS';
                  
END_GET
END_PROPERTY
END_FUNCTION_BLOCK

FUNCTION_BLOCK Charger EXTENDS NonOperationalParticleSet
  VAR CONSTANT
    cMaximumChargeLevel : t_percentage := 1.0;
    cDefaultChargeLevel : t_percentage := 0.95;
    cMinimumChargeLevel : t_percentage := 0.1;
    cTargetChargeLevelHysteresis : t_percentage := 0.01;
    cManualChargingCurrentTarget : REAL := 5.0;
    cManualChargingVoltageTarget : REAL := 130.0;
  END_VAR
  VAR
    lVREnableManualNotBMSCharging : ValueReferenceBool;
    lEnableManualNotBMSCharging : BOOL := FALSE;
    lVRManualChargingCurrentTarget : ValueReferenceReal;
    lManualChargingCurrentTarget : REAL := cManualChargingCurrentTarget;
    lVRManualChargingVoltageTarget : ValueReferenceReal;
    lManualChargingVoltageTarget : REAL := cManualChargingVoltageTarget;
    lAlarmChargerOBCError : ReportableSystemControl;
    lCausalChargerStandby : ReportableSystemControl;
    lCausalChargerConnected : ReportableSystemControl;
    lCausalChargerDisconnected : ReportableCausal;
    lTargetBMSChargeState : t_bms_charge_state;
    lRequestedBMSChargeState : t_bms_charge_state;
    lCurrentBMSChargeState : t_bms_charge_state;
    lRequestedOBCState : t_obc_state;
    lCurrentOBCState : t_obc_state;
    lPreviousOBCState : t_obc_state := cOBCStateDisconnected;
    lChargingCurrentTarget : REAL;
    lChargingVoltageTarget : REAL;
    lTargetChargeLevel : t_percentage := cDefaultChargeLevel;
    lChargerDiagnostic : t_charger_diagnostic;
  END_VAR

            ;
          

METHOD _operator
                  IF ((lCurrentOBCState<>lPreviousOBCState) AND
	(lPreviousOBCState=cOBCStateDisconnected)) THEN
	gSystemPrimary.BMS.resetSOCRecovery();
END_IF
lPreviousOBCState := lCurrentOBCState;

gSystemPrimary.SystemState.ChargingEnabled := (lCurrentOBCState<>cOBCStateDisconnected);

CASE (lCurrentOBCState) OF
	cOBCStateDisconnected:
		IF (gSystemPrimary.SystemState.State=cSystemStateCharging) THEN
			lCausalChargerDisconnected.trigger(FALSE);
			gSystemPrimary.SystemState.transitionForceMax(cSystemStatePreparing,ADR(lCausalChargerDisconnected),lCausalChargerDisconnected.Override);
		END_IF
		lChargingCurrentTarget := 0.0;
		lChargingVoltageTarget := 0.0;
	
		lChargerDiagnostic := cChargingDiagnosticDisconnected;
		
		IF (NOT(Operational)) THEN
			lChargerDiagnostic := cChargingDiagnosticNotOperational;
		END_IF

	cOBCStateError:
		lAlarmChargerOBCError.trigger(FALSE);
		lChargerDiagnostic := cChargingDiagnosticConnectedError;

 cOBCStateStandby:
 		lCausalChargerStandby.trigger(FALSE);
		lChargerDiagnostic := cChargingDiagnosticConnectedStandby;
		
	cOBCStateCharging:
		lCausalChargerConnected.trigger(FALSE);
		lChargerDiagnostic := cChargingDiagnosticConnected;
END_CASE

IF (gSystemPrimary.SystemState.State<>cSystemStateCharging) THEN
	lRequestedOBCState := cOBCStateStandby;
	lRequestedBMSChargeState := cBMSChargeStateShutdown;

	lChargingCurrentTarget := 0.0;
	lChargingVoltageTarget := 0.0;
	
	lChargerDiagnostic := cChargingDiagnosticNotInChargingState;
	
	RETURN;
END_IF

IF ((gSystemPrimary.BMS.SOCMax>=lTargetChargeLevel) OR
	((lCurrentBMSChargeState=cBMSChargeStateShutdown) AND
	(gSystemPrimary.BMS.SOCMax>=(lTargetChargeLevel-cTargetChargeLevelHysteresis)))) THEN
	lRequestedOBCState := cOBCStateStandby;
	lRequestedBMSChargeState := cBMSChargeStateShutdown;
	
	lChargingCurrentTarget := 0.0;
	lChargingVoltageTarget := 0.0;
	
	lChargerDiagnostic := cChargingDiagnosticTargetSOCReached;
	
	RETURN;
END_IF

lRequestedBMSChargeState := lTargetBMSChargeState;
IF (lCurrentBMSChargeState=cBMSChargeStateShutdown) THEN
	lChargingCurrentTarget := 0.0;
	lChargingVoltageTarget := 0.0; // foobar, make sure this cannot be overwritten
	
	lChargerDiagnostic := cChargingDiagnosticBMSShutdown;
	
	RETURN;
END_IF

IF (lChargingCurrentTarget<>0.0) THEN
	lChargerDiagnostic := cChargingDiagnosticConnectedCharging;
END_IF

lRequestedOBCState := cOBCStateCharging;


                
END_METHOD

METHOD initialize
                  lVREnableManualNotBMSCharging.initializeValueReference(lEnableManualNotBMSCharging,NopSelf,'EnblManualChrg','Enable manual charging control','',cValueStyleParameter);
lVRManualChargingCurrentTarget.initializeValueReference(lManualChargingCurrentTarget,NopSelf,'ManualChrgCurr','Manual charging current','amps',cValueStyleParameter);
lVRManualChargingVoltageTarget.initializeValueReference(lManualChargingVoltageTarget,NopSelf,'ManualChrgVolt','Manual charging voltage','volts',cValueStyleParameter);

lAlarmChargerOBCError.initializeState(NopSelf,'',cACChargerOBCError);
lAlarmChargerOBCError.Control := cSystemControlStop;
lAlarmChargerOBCError.AllowableSystemState := cSystemStateCharging;

lCausalChargerStandby.initializeState(NopSelf,'',cCCChargerStandby);
lCausalChargerStandby.Control := cSystemControlStop;
lCausalChargerStandby.AllowableSystemState := cSystemStateCharging;

lCausalChargerConnected.initializeState(NopSelf,'',cCCChargerConnected);
lCausalChargerConnected.Control := cSystemControlStop;
lCausalChargerConnected.AllowableSystemState := cSystemStateCharging;

lCausalChargerDisconnected.initializeState(NopSelf,'',cCCChargerDisconnected);

SUPER^.initialize();
SubSystem := cSubsystemBattery;

                
END_METHOD

METHOD operator
                  lCurrentBMSChargeState := gSystemPrimary.BMS.CurrentBMSChargeState;
lChargingCurrentTarget := gSystemPrimary.BMS.ChargingCurrentTarget;
lChargingVoltageTarget := gSystemPrimary.BMS.ChargingVoltageTarget;

_operator();

gSystemPrimary.BMS.RequestedBMSChargeState := lRequestedBMSChargeState;

IF (lEnableManualNotBMSCharging) THEN
	lRequestedOBCState := cOBCStateCharging;
	lChargingCurrentTarget := lManualChargingCurrentTarget;
	lChargingVoltageTarget := lManualChargingVoltageTarget;
END_IF

                
END_METHOD

(* {attribute 'monitoring' := 'call'} *)
PROPERTY ChargerDiagnostic : t_charger_diagnostic
GET
                    ChargerDiagnostic := lChargerDiagnostic;
                  
END_GET
END_PROPERTY

PROPERTY ChargingCurrentTarget : REAL
GET
                    ChargingCurrentTarget := lChargingCurrentTarget;

                  
END_GET
SET
                    lChargingCurrentTarget := ChargingCurrentTarget;
                  
END_SET
END_PROPERTY

PROPERTY ChargingVoltageTarget : REAL
GET
                    ChargingVoltageTarget := lChargingVoltageTarget;

                  
END_GET
SET
                    lChargingVoltageTarget := ChargingVoltageTarget;

                  
END_SET
END_PROPERTY

PROPERTY CurrentBMSChargeState : t_bms_charge_state
GET
                    CurrentBMSChargeState := lCurrentBMSChargeState;

                  
END_GET
SET
                    lCurrentBMSChargeState := CurrentBMSChargeState;
                  
END_SET
END_PROPERTY

PROPERTY CurrentOBCState : t_obc_state
GET
                    CurrentOBCState := lCurrentOBCState;

                  
END_GET
END_PROPERTY

PROPERTY Operational : BOOL
GET
                    Operational := false;
                  
END_GET
END_PROPERTY

PROPERTY RequestedBMSChargeState : t_bms_charge_state
GET
                    RequestedBMSChargeState := lRequestedBMSChargeState;

                  
END_GET
SET
                    lRequestedBMSChargeState := RequestedBMSChargeState;
                  
END_SET
END_PROPERTY

PROPERTY RequestedOBCState : t_obc_state
GET
                    RequestedOBCState := lRequestedOBCState;
                  
END_GET
END_PROPERTY

PROPERTY TargetBMSChargeState : t_bms_charge_state
GET
                    TargetBMSChargeState := lTargetBMSChargeState;
                  
END_GET
END_PROPERTY

PROPERTY TargetChargeLevel : t_percentage
GET
                    TargetChargeLevel := lTargetChargeLevel;
                  
END_GET
SET
                    lTargetChargeLevel := TargetChargeLevel;

lTargetChargeLevel := MIN(lTargetChargeLevel,cMaximumChargeLevel);
lTargetChargeLevel := MAX(lTargetChargeLevel,cMinimumChargeLevel);


                  
END_SET
END_PROPERTY

PROPERTY TypeToken : t_medium_string
GET
                    TypeToken := 'Charger';
                  
END_GET
END_PROPERTY
END_FUNCTION_BLOCK

FUNCTION_BLOCK ChargerA EXTENDS Charger
  VAR
    lControllerChargerA : REFERENCE TO ControllerCharger;
  END_VAR

            ;
          

METHOD initialize
                  IF (NOT(__ISVALIDREF(lControllerChargerA))) THEN
	gCodeErrorHandler(pMessage:=CONCAT('null reference in ',lIdentity));
END_IF

SUPER^.initialize();



                
END_METHOD

METHOD operator
                  lTargetBMSChargeState := cBMSChargeStateAC;

lCurrentOBCState := lControllerChargerA.CurrentOBCState;

SUPER^.operator();

lControllerChargerA.RequestedOBCState := lRequestedOBCState;
lControllerChargerA.ChargingCurrentMax := lChargingCurrentTarget;
lControllerChargerA.ChargingVoltageMax := lChargingVoltageTarget;

                
END_METHOD

METHOD initializeCharger
  VAR_INPUT
    controllerCharger : REFERENCE TO ControllerCharger;
  END_VAR
                  lControllerChargerA REF= controllerCharger;
                
END_METHOD

PROPERTY Operational : BOOL
GET
                    Operational := lControllerChargerA.Operational;
                  
END_GET
END_PROPERTY
END_FUNCTION_BLOCK

FUNCTION_BLOCK ChargerABC EXTENDS Charger
  VAR
    lControllerChargerA : REFERENCE TO ControllerCharger;
    lControllerChargerB : REFERENCE TO ControllerCharger;
    lControllerChargerC : REFERENCE TO ControllerCharger;
  END_VAR

            ;
          

METHOD initialize
                  IF ((NOT(__ISVALIDREF(lControllerChargerA))) OR
	(NOT(__ISVALIDREF(lControllerChargerB))) OR
	(NOT(__ISVALIDREF(lControllerChargerC)))) THEN
	gCodeErrorHandler(pMessage:=CONCAT('null reference in ',lIdentity));
END_IF

SUPER^.initialize();

                
END_METHOD

METHOD operator
                  lTargetBMSChargeState := cBMSChargeStateAC;

lCurrentOBCState := lControllerChargerA.CurrentOBCState;

SUPER^.operator();

lControllerChargerA.RequestedOBCState := lRequestedOBCState;
lControllerChargerA.ChargingCurrentMax := lChargingCurrentTarget/3.0;
lControllerChargerA.ChargingVoltageMax := lChargingVoltageTarget;

lControllerChargerB.RequestedOBCState := lRequestedOBCState;
lControllerChargerB.ChargingCurrentMax := lChargingCurrentTarget/3.0;
lControllerChargerB.ChargingVoltageMax := lChargingVoltageTarget;

lControllerChargerC.RequestedOBCState := lRequestedOBCState;
lControllerChargerC.ChargingCurrentMax := lChargingCurrentTarget/3.0;
lControllerChargerC.ChargingVoltageMax := lChargingVoltageTarget;

                
END_METHOD

METHOD initializeCharger
  VAR_INPUT
    controllerChargerA : REFERENCE TO ControllerCharger;
    controllerChargerB : REFERENCE TO ControllerCharger;
    controllerChargerC : REFERENCE TO ControllerCharger;
  END_VAR
                  lControllerChargerA REF= controllerChargerA;
lControllerChargerB REF= controllerChargerB;
lControllerChargerC REF= controllerChargerC;
                
END_METHOD

PROPERTY Operational : BOOL
GET
                    Operational := lControllerChargerA.Operational;
                  
END_GET
END_PROPERTY

PROPERTY TypeToken : t_medium_string
GET
                    TypeToken := 'ChargerABC';
                  
END_GET
END_PROPERTY
END_FUNCTION_BLOCK

FUNCTION_BLOCK ControllerBMS EXTENDS ControllerSlavePLC
  VAR CONSTANT
    cChargingCurrentTargetDefault : REAL := 40.0;  (* foobar is this machine specific? *)
    cAvailabilityLimitedSevere : t_percentage := 0.5;
    cChargeCurrentLimit : REAL := 450;
    cDischargeCurrentLimit : REAL := 450;
    cContextSize : USINT := 8;
  END_VAR
  VAR
    lVROverrideBMSChargeStateControl : ValueReferenceBool;
    lOverrideBMSChargeStateControl : BOOL := TRUE;  (* foobar why is this defaulting to true, CATL bug *)
    lAlarmChargeAvailabilityLimited : ReportableAlarm;
    lAlarmChargeAvailabilityLimitedSevere : ReportableAlarm;
    lAlarmDischargeAvailabilityLimited : ReportableAlarm;
    lAlarmDischargeAvailabilityLimitedSevere : ReportableAlarm;
    lAlarmBMSRequestDisconnect : ReportableAlarmEscalating;
    lAlarmBMSFault : ReportableAlarm;
    lPeripheral : PeripheralPrimary;
    lRequestedBMSState : ValueObjectEnumTypeOutputReferenceUSINT;  (* lDischargeEnergy: EnergyMetric; foostrip lChargeEnergy: EnergyMetric; foostrip *)
    lCurrentTMSState : ValueObjectEnumTypeOutputReferenceUSINT;
    lRequestedBMSChargeState : ValueObjectEnumTypeOutputReferenceUSINT;
    lCurrentCoolantTemperature : ValueObjectRealScaledOffsetOutputReferenceUSINT;
    lCurrentBMSState : ValueObjectEnumTypeInputReferenceUSINT;
    lRequestedTMSState : ValueObjectEnumTypeInputReferenceUSINT;
    lCurrentBMSChargeState : ValueObjectEnumTypeInputReferenceUSINT;
    lBalancing : ValueObjectBoolInputReferenceUSINT;
    lRequestDisconnect : ValueObjectBoolInputReferenceUSINT;
    lFaultCharger : ValueObjectBoolInputReferenceUSINT;
    lFaultContactor : ValueObjectBoolInputReferenceUSINT;
    lFaultLevel : ValueObjectEnumTypeInputReferenceUSINT;
    lPackCurrent : ValueObjectRealScaledOffsetInputReferenceUINT;  (* lGateway2PLCState1: ValueObjectUSINTGateway2PLCState1; lGateway2PLCState2: ValueObjectUSINTGateway2PLCState2; *)
    lPackChargeCurrentLimit : ValueObjectRealScaledOffsetInputReferenceUINT;
    lPackDischargeCurrentLimit : ValueObjectRealScaledOffsetInputReferenceUINT;
    lPackVoltage : ValueObjectRealScaledOffsetInputReferenceUINT;
    lPackAverageTemperature : ValueObjectRealScaledOffsetInputReferenceUSINT;
    lPackMaxTemperature : ValueObjectRealScaledOffsetInputReferenceUSINT;
    lPackMinTemperature : ValueObjectRealScaledOffsetInputReferenceUSINT;
    lPackSOC : ValueObjectPercentageScaledOffsetInputReferenceUSINT;
    lPackSOH : ValueObjectPercentageScaledOffsetInputReferenceUSINT;
    lPackChargingCurrentTarget : ValueObjectRealScaledOffsetInputReferenceUINT;
    lPackChargingVoltageTarget : ValueObjectRealScaledOffsetInputReferenceUINT;
    lPackCoolantTemperatureTarget : ValueObjectRealScaledOffsetInputReferenceUSINT;
    lPackTotalChargeEnergy : ValueObjectRealReference3xUSINT;
    lPackTotalDischargeEnergy : ValueObjectRealReference3xUSINT;
    lPackFaultNumber : ValueObjectUSINTInputReferenceUSINT;
    lPackFaultCode : ValueObjectUSINTInputReferenceUSINT;
    lChargeAvailability : t_percentage;  (* lPackFaultByte1: ValueBitsBMSByte1; lPackFaultByte2: ValueBitsBMSByte2; lPackFaultByte3: ValueBitsBMSByte3; lPackFaultByte4: ValueBitsBMSByte4; lPackFaultByte5: ValueBitsBMSByte5; lPackFaultByte6: ValueBitsBMSByte6; lPackFaultByte7: ValueBitsBMSByte7; lPackFaultByte8: ValueBitsBMSByte8; lPackFaultByte9: ValueBitsBMSByte9; lPackFaultByte10: ValueBitsBMSByte10; lPackFaultByte11: ValueBitsBMSByte11; *)
    lDischargeAvailability : t_percentage;
    lFaultNumber : USINT;
    lFaultCode : t_bms_fault_id;
    lFaults : ARRAY[0..7] OF t_bms_fault_id;
    lContextIndex : USINT;
    lContextPtr : POINTER TO BYTE;
    lContext : LWORD;
    lCollected : BOOL;
  END_VAR

            ;
          

METHOD initialize
                  lAlarmBMSRequestDisconnect.initializeState(NopSelf,'',cACBMSRequestDisconnect);
lAlarmBMSRequestDisconnect.Life := 10;
lAlarmBMSRequestDisconnect.InitialSeverity := cSeverityError;
lAlarmBMSRequestDisconnect.SeverityWarningTimeout := T#0S;
lAlarmBMSRequestDisconnect.SeverityErrorTimeout := T#5S;
lAlarmBMSRequestDisconnect.SeverityCriticalTimeout := T#25S;

lAlarmChargeAvailabilityLimited.initializeState(NopSelf,'',cBMSChargeAvailabilityLimited);
lAlarmChargeAvailabilityLimited.Life := 10;

lAlarmChargeAvailabilityLimitedSevere.initializeState(NopSelf,'',cBMSChargeAvailabilityLimitedSevere);
lAlarmChargeAvailabilityLimitedSevere.Life := 10;

lAlarmDischargeAvailabilityLimited.initializeState(NopSelf,'',cBMSDischargeAvailabilityLimited);
lAlarmDischargeAvailabilityLimited.Life := 10;

lAlarmDischargeAvailabilityLimitedSevere.initializeState(NopSelf,'',cBMSDischargeAvailabilityLimitedSevere);
lAlarmDischargeAvailabilityLimitedSevere.Life := 10;

lAlarmBMSFault.initializeState(NopSelf,'',cACBMSFault);

lVROverrideBMSChargeStateControl.initializeValueReference(lOverrideBMSChargeStateControl,NopSelf,'OvrdChrgSttCntrl','Override charging control by the BMS','',cValueStyleParameter);

// foostrip lDischargeEnergy.Name := 'DischargeEnergy';
//registerNonOperational(ADR(lDischargeEnergy));
//lChargeEnergy.Name := 'ChargeEnergy';
//registerNonOperational(ADR(lChargeEnergy));

lRequestedBMSState.MergeOutput := FALSE;
lRequestedBMSState.Index := 0;
lRequestedBMSState.EnumType := cEnumTypeBMSState;
lRequestedBMSState.initializeValueObjectOp(OpSelf,'ReqBMSStt','Requested BMS state','',cValueStyleConfigurable);

lCurrentTMSState.MergeOutput := TRUE;
lCurrentTMSState.Index := 2;
lCurrentTMSState.EnumType := cEnumTypeTMSState;
lCurrentTMSState.initializeValueObjectOp(OpSelf,'CurrTMSStt','Current TMS state','',cValueStyleConfigurable);

lRequestedBMSChargeState.MergeOutput := TRUE;
lRequestedBMSChargeState.Index := 4;
lRequestedBMSChargeState.EnumType := cEnumTypeBMSChargeState;
lRequestedBMSChargeState.initializeValueObjectOp(OpSelf,'ReqBMSChrgStt','Requested BMS charge state','',cValueStyleConfigurable);

lCurrentBMSState.Index := 1;
lCurrentBMSState.Length := 2;
lCurrentBMSState.EnumType := cEnumTypeBMSState;
lCurrentBMSState.initializeValueObjectOp(OpSelf,'CurrBMSStt','Current BMS state','',cValueStyleConfigurable);

lRequestedTMSState.Index := 3;
lRequestedTMSState.Length := 2;
lRequestedTMSState.EnumType := cEnumTypeTMSState;
lRequestedTMSState.initializeValueObjectOp(OpSelf,'ReqTMSStt','Requested TMS state','',cValueStyleConfigurable);

lCurrentBMSChargeState.Index := 5;
lCurrentBMSChargeState.Length := 2;
lCurrentBMSChargeState.EnumType := cEnumTypeBMSChargeState;
lCurrentBMSChargeState.initializeValueObjectOp(OpSelf,'CurrBMSChrgStt','Current BMS charge state','',cValueStyleConfigurable);
	
lCurrentCoolantTemperature.Scaling := 1.0;
lCurrentCoolantTemperature.Offset := -40.0;
lCurrentCoolantTemperature.initializeValueObjectOp(OpSelf,'CurrCoolantTemp','Current coolant temperature','',cValueStyleConfigurable);

lBalancing.Index := 0;
lBalancing.initializeValueObjectOp(OpSelf,'Balancing','Current BMS balancing status','',cValueStyleConfigurable);

lRequestDisconnect.Index := 7;
lRequestDisconnect.initializeValueObjectOp(OpSelf,'RqstDisconnect','Current BMS disconnect request','',cValueStyleConfigurable);

lFaultCharger.Index := 4;
lFaultCharger.initializeValueObjectOp(OpSelf,'FaultCharger','Current BMS charger fault state','',cValueStyleConfigurable);
lFaultContactor.Index := 3;
lFaultContactor.initializeValueObjectOp(OpSelf,'FaultContactor','Current BMS contactor fault state','',cValueStyleConfigurable);

lFaultLevel.Index := 0;
lFaultLevel.Length := 3;
lFaultLevel.EnumType := cEnumTypeBMSFaultLevel;
lFaultLevel.initializeValueObjectOp(OpSelf,'FaultLevel','Current BMS fault level','',cValueStyleConfigurable);
	
lPackCurrent.Scaling := 0.1;
lPackCurrent.Offset := -1000.0;
lPackCurrent.initializeValueObjectOp(OpSelf,'Current','Current BMS current','amps',cValueStyleConfigurable);

lPackChargeCurrentLimit.Scaling := 0.1;
lPackChargeCurrentLimit.Offset := 0.0;
lPackChargeCurrentLimit.initializeValueObjectOp(OpSelf,'ChrgCurrLmt','Current BMS charge current limit','amps',cValueStyleConfigurable);

lPackDischargeCurrentLimit.Scaling := 0.1;
lPackDischargeCurrentLimit.Offset := 0.0;
lPackDischargeCurrentLimit.initializeValueObjectOp(OpSelf,'DschrgCurrLmt','Current BMS discharge current limit','amps',cValueStyleConfigurable);

lPackVoltage.Scaling := 0.1;
lPackVoltage.Offset := 0.0;
lPackVoltage.initializeValueObjectOp(OpSelf,'Voltage','Current BMS voltage','volts',cValueStyleConfigurable);

lPackAverageTemperature.Scaling := 1.0;
lPackAverageTemperature.Offset := -40.0;
lPackAverageTemperature.initializeValueObjectOp(OpSelf,'AverageTemp','Current BMS average temperature','celcius',cValueStyleConfigurable);

lPackMaxTemperature.Scaling := 1.0;
lPackMaxTemperature.Offset := -40.0;
lPackMaxTemperature.initializeValueObjectOp(OpSelf,'MaxTemp','Current BMS max temperature','celcius',cValueStyleConfigurable);

lPackMinTemperature.Scaling := 1.0;
lPackMinTemperature.Offset := -40.0;
lPackMinTemperature.initializeValueObjectOp(OpSelf,'MinTemp','Current BMS min temperature','celcius',cValueStyleConfigurable);
	
lPackSOC.Scaling := 0.004;
lPackSOC.Offset := 0.0;	
lPackSOC.initializeValueObjectOp(OpSelf,'SOC','Current BMS State-of-Charge','',cValueStyleConfigurable);

lPackSOH.Scaling := 0.004;
lPackSOH.Offset := 0.0;	
lPackSOH.initializeValueObjectOp(OpSelf,'SOH','Current BMS State-of-Health','',cValueStyleConfigurable);

lPackChargingCurrentTarget.OverrideValue := cChargingCurrentTargetDefault;
lPackChargingCurrentTarget.Scaling := 0.1;
lPackChargingCurrentTarget.Offset := 0.0;	
lPackChargingCurrentTarget.initializeValueObjectOp(OpSelf,'ChrgCurrTrgt','Target BMS charge current','amps',cValueStyleConfigurable);

lPackChargingVoltageTarget.Scaling := 0.1;
lPackChargingVoltageTarget.Offset := 0.0;	
lPackChargingVoltageTarget.initializeValueObjectOp(OpSelf,'ChrgVoltTrgt','Target BMS charge voltage','volts',cValueStyleConfigurable);

lPackCoolantTemperatureTarget.Scaling := 0.4;
lPackCoolantTemperatureTarget.Offset := 0.0;	
lPackCoolantTemperatureTarget.initializeValueObjectOp(OpSelf,'CoolantTempTrgt','Target BMS coolant temperature','celcius',cValueStyleConfigurable);

lPackTotalChargeEnergy.initializeValueObjectOp(OpSelf,'TtlChrgEnergy','BMS cumulative charge energy','kJ',cValueStyleConfigurable);
lPackTotalDischargeEnergy.initializeValueObjectOp(OpSelf,'TtlDschrgEnergy','BMS cumulative discharge energy','kJ',cValueStyleConfigurable);

lPackFaultNumber.initializeValueObjectOp(OpSelf,'FaultNumber','Current BMS fault count','',cValueStyleConfigurable);
lPackFaultCode.initializeValueObjectOp(OpSelf,'FaultCode','Current BMS fault code','',cValueStyleConfigurable);

SUPER^.initialize();
SubSystem := cSubsystemBattery;

lPeripheral.initialize();

lAlarmCANOpenSlaveNotOperational.InitialSeverity := cSeverityNone;
lAlarmCANOpenSlaveNotOperational.SeverityWarningTimeout := T#250MS;
lAlarmCANOpenSlaveNotOperational.SeverityErrorTimeout := T#1S;
lAlarmCANOpenSlaveNotOperational.SeverityCriticalTimeout := T#5S;

lAlarmCANOpenSlaveAllowableUp.AllowableSystemState := cSystemStatePreparing;
lAlarmCANOpenSlaveAllowableUp.UpperSystemStateScope := cSystemStatePreparing;
lAlarmCANOpenSlaveAllowableUp.LowerSystemStateScope := cSystemStatePreparing;

lStartSystemStateScope := t_system_state.cSystemStatePreparing;
lOperationalSystemStateScopeLower := t_system_state.cSystemStateCharging;
lModulationSystemStateScope := t_system_state.cSystemStateCharging;

lModulationSeverity := cSeverityError;

lEnableValidTransmissions := TRUE;
lEnableDetectionTPDO := TRUE;
lEnableNMTDetectionTPDO := TRUE;
lEnableNMTOverrideTPDO := TRUE;

lContextPtr := ADR(lContext);
lContextIndex := 0;
lFaultNumber := 0;
lFaultCode := 0;
lCollected := false;

                
END_METHOD

METHOD operator
  VAR
    fault : t_bms_fault_id;
    ptr : POINTER TO BYTE;
    i : USINT;
  END_VAR
                  SUPER^.operator();

lPeripheral.operator();

IF (NOT(ValidTransmissions)) THEN
	lCurrentBMSState.Value := cBMSStateShutdown;
END_IF

IF (lCurrentBMSState.Value<cBMSStateDisconnected) THEN
	lRequestedTMSState.Value := cTMSStateShutdown;
	lCurrentBMSChargeState.Value := cBMSChargeStateShutdown;
	lRequestDisconnect.Value := FALSE;

	lFaultLevel.Value := cBMSFaultLevelNone;
	lPackFaultNumber.Value := 0;
	lPackFaultCode.Value := 0;
	lFaultCharger.Value := FALSE;
	lFaultContactor.Value := FALSE;

	lPackSOC.Value := 0.0;
	lPackSOH.Value := 1.0;
	
	lPackCurrent.Value:= 0.0;
	lPackChargeCurrentLimit.Value := 0.0;
	lPackDischargeCurrentLimit.Value := 0.0;
	lPackVoltage.Value := 0.0;
		
	RETURN;
END_IF

IF ((gSystemPrimary.SystemState.State>cSystemStatePreparing) AND
	(RequestDisconnect)) THEN
	lAlarmBMSRequestDisconnect.trigger(FALSE);
	
	IF (lAlarmBMSRequestDisconnect.Severity>=cSeverityCritical) THEN
		lRequestedBMSState.Value := cBMSStateDisconnected;
	END_IF
END_IF

lChargeAvailability := lPackChargeCurrentLimit.Value/cChargeCurrentLimit;
IF (lChargeAvailability<cAvailabilityLimitedSevere) THEN
	lAlarmChargeAvailabilityLimitedSevere.trigger(FALSE);
ELSIF (lChargeAvailability<1.0) THEN
	lAlarmChargeAvailabilityLimited.trigger(FALSE);
END_IF

lDischargeAvailability := lPackChargeCurrentLimit.Value/cDischargeCurrentLimit;
IF (lDischargeAvailability<cAvailabilityLimitedSevere) THEN
	lAlarmDischargeAvailabilityLimitedSevere.trigger(FALSE);
ELSIF (lDischargeAvailability<1.0) THEN
	lAlarmDischargeAvailabilityLimited.trigger(FALSE);
END_IF

//foostrip lChargeEnergy.integrate(PackChargeCurrent,PackVoltage);
//lDischargeEnergy.integrate(PackDischargeCurrent,PackVoltage);

IF (lPackFaultNumber.Value<>lFaultNumber) THEN
	lFaultNumber := lPackFaultNumber.Value;
	lFaultCode := 0;
	lContextIndex := 0;
	lContext := 0;
	lCollected := FALSE;
	
	for i:= 0 to 7 do
		lFaults[i] := 0;
	END_FOR
END_IF

IF (lFaultNumber=0) THEN
	RETURN;
END_IF

IF (lFaultCode<>lPackFaultCode.Value) THEN
	lFaultCode := lPackFaultCode.Value;
	
	IF (lContextIndex<cContextSize) THEN
		lContextPtr := ADR(lContext);
		lContextPtr := lContextPtr + lContextIndex;
	
		lContextPtr^ := INT_TO_BYTE(lFaultCode);
		lFaults[lContextIndex] := lFaultCode;
	END_IF

	lContextIndex := lContextIndex + 1;
END_IF

IF (lContextIndex>=lFaultNumber) THEN
	lContextIndex := 0;
	lCollected := TRUE;
END_IF

IF (lCollected) THEN
	lAlarmBMSFault.triggerWithContext(lContext);
END_IF


                
END_METHOD

METHOD initializeBMS
  VAR_INPUT
    gateway2PLCState1 : REFERENCE TO USINT;
    gateway2PLCState2 : REFERENCE TO USINT;
    packCurrent : REFERENCE TO UINT;
    packChargeCurrentLimit : REFERENCE TO UINT;
    packDischargeCurrentLimit : REFERENCE TO UINT;
    packVoltage : REFERENCE TO UINT;
    packAverageTemperature : REFERENCE TO USINT;
    packMaxTemperature : REFERENCE TO USINT;
    packMinTemperature : REFERENCE TO USINT;
    packSOC : REFERENCE TO USINT;
    packSOH : REFERENCE TO USINT;
    packChargingCurrentTarget : REFERENCE TO UINT;
    packChargingVoltageTarget : REFERENCE TO UINT;
    packCoolantTemperatureTarget : REFERENCE TO USINT;
    packTotalChargeEnergyA : REFERENCE TO USINT;
    packTotalChargeEnergyB : REFERENCE TO USINT;
    packTotalChargeEnergyC : REFERENCE TO USINT;
    packTotalDischargeEnergyA : REFERENCE TO USINT;
    packTotalDischargeEnergyB : REFERENCE TO USINT;
    packTotalDischargeEnergyC : REFERENCE TO USINT;
    packFaultNumber : REFERENCE TO USINT;
    packFaultCode : REFERENCE TO USINT;
    pLC2GatewayState : REFERENCE TO USINT;
    coolantTemperature : REFERENCE TO USINT;
  END_VAR
                  lCurrentBMSState.InputReference REF= gateway2PLCState1;
lRequestedTMSState.InputReference REF= gateway2PLCState1;
lCurrentBMSChargeState.InputReference REF= gateway2PLCState1;

lBalancing.InputReference REF= gateway2PLCState1;
lRequestDisconnect.InputReference REF= gateway2PLCState1;

lFaultCharger.InputReference REF= gateway2PLCState2;
lFaultContactor.InputReference REF= gateway2PLCState2;
lFaultLevel.InputReference REF= gateway2PLCState2;

lPackCurrent.InputReference REF= packCurrent;
lPackChargeCurrentLimit.InputReference REF= packChargeCurrentLimit;
lPackDischargeCurrentLimit.InputReference REF= packDischargeCurrentLimit;
lPackVoltage.InputReference REF= packVoltage;

lPackAverageTemperature.InputReference REF= packAverageTemperature;
lPackMaxTemperature.InputReference REF= packMaxTemperature;
lPackMinTemperature.InputReference REF= packMinTemperature;

lPackSOC.InputReference REF= packSOC;
lPackSOH.InputReference REF= packSOH;

lPackChargingCurrentTarget.InputReference REF= packChargingCurrentTarget;
lPackChargingVoltageTarget.InputReference REF= packChargingVoltageTarget;
lPackCoolantTemperatureTarget.InputReference REF= packCoolantTemperatureTarget;

lPackTotalChargeEnergy.InputReferenceA REF= packTotalChargeEnergyA;
lPackTotalChargeEnergy.InputReferenceB REF= packTotalChargeEnergyB;
lPackTotalChargeEnergy.InputReferenceC REF= packTotalChargeEnergyC;

lPackTotalDischargeEnergy.InputReferenceA REF= packTotalDischargeEnergyA;
lPackTotalDischargeEnergy.InputReferenceB REF= packTotalDischargeEnergyB;
lPackTotalDischargeEnergy.InputReferenceC REF= packTotalDischargeEnergyC;

lPackFaultNumber.InputReference REF= packFaultNumber;
lPackFaultCode.InputReference REF= packFaultCode;

lRequestedBMSState.OutputReference REF= pLC2GatewayState;
lCurrentTMSState.OutputReference REF= pLC2GatewayState;
lRequestedBMSChargeState.OutputReference REF= pLC2GatewayState;

lCurrentCoolantTemperature.OutputReference REF= coolantTemperature;	
                
END_METHOD

PROPERTY Balancing : BOOL
GET
                    Balancing := lBalancing.Value;
                  
END_GET
END_PROPERTY

PROPERTY CurrentBMSChargeState : t_bms_charge_state
GET
                    lPackChargingCurrentTarget.Override := FALSE;

IF (Operational) THEN
	IF ((RequestedBMSChargeState<>cBMSChargeStateShutdown) AND (lOverrideBMSChargeStateControl)) THEN
		CurrentBMSChargeState := RequestedBMSChargeState;
		lPackChargingCurrentTarget.Override := TRUE;
	ELSE
		CurrentBMSChargeState := lCurrentBMSChargeState.Value;
	END_IF
ELSE
	CurrentBMSChargeState := cBMSChargeStateShutdown;	
END_IF

                  
END_GET
END_PROPERTY

PROPERTY CurrentBMSState : t_bms_state
GET
                    IF (Operational) THEN
	CurrentBMSState := lCurrentBMSState.Value;
ELSE
	CurrentBMSState := cBMSStateShutdown;	
END_IF
                  
END_GET
END_PROPERTY

PROPERTY CurrentCoolantTemperature : REAL
GET
                    CurrentCoolantTemperature := lCurrentCoolantTemperature.Value;
                  
END_GET
SET
                    lCurrentCoolantTemperature.Value := CurrentCoolantTemperature;
                  
END_SET
END_PROPERTY

PROPERTY CurrentTMSState : t_tms_state
GET
                    CurrentTMSState := lCurrentTMSState.Value;
                  
END_GET
SET
                    lCurrentTMSState.Value := CurrentTMSState;
                  
END_SET
END_PROPERTY

PROPERTY FaultCharger : BOOL
GET
                    IF (Operational) THEN
	FaultCharger := lFaultCharger.Value;
ELSE
	FaultCharger := FALSE;	
END_IF
                  
END_GET
END_PROPERTY

